// TIA Portal V19 export
FUNCTION_BLOCK "JB_FB"   // FB68, LAD
TITLE = JUNCTION BENCH WELDER
// stored: MemoryReserve 100, SetENOAutomatically false
   VAR_INPUT
      AreaInterface : "AreaInterface";
      ZSI : "udt_ZoneSafetyInterface";
      DSI : Struct
         Torch : "udt_DeviceSafetyInterface";
         ClampEntry : "udt_DeviceSafetyInterface";
         ClampExit : "udt_DeviceSafetyInterface";
         CutHead : "udt_DeviceSafetyInterface";
         PinchRoll_Feed : "udt_DeviceSafetyInterface";
         PinchRoll_Lift : "udt_DeviceSafetyInterface";
      END_STRUCT;
      Drive : Struct
         Torch : "TAx_DriveInterface";
         Picnhroll_Feed : "TAx_DriveInterface";
      END_STRUCT;
      HWID : Struct
         Torch_TEL1 : HW_SUBMODULE;
         TorchEnc_IO : HW_SUBMODULE;
         Pinchroll_Feed_TEL1 : HW_SUBMODULE;
      END_STRUCT;
      DataIn : Struct
         WeldingCycle_AI_Potentiometer : Int;
         WeldingCycle_Pb_Stop : Bool;
         WeldingCycle_Pb_Start : Bool;
         WeldingCycle_Pb_StartStop : Bool;
         Welder_Pb_Man : Bool;
         CutHead_PbCycle : Bool;
         SAFETY_DeadMan_PB : Bool;   // Pulsante presenza uomo SAFTEY
         Torch : "Positioning_DOL_Machine_DataIn";
         ClampEntry : "ValveMachine_DataIn";
         ClampExit : "ValveMachine_DataIn";
         CutHead : "ValveMachine_DataIn";
         PinchRoll_Feed : "SpeedMachine_DataIn";
         PinchRoll_Lift : "ValveMachine_DataIn";
      END_STRUCT;
      CIn : Struct
         Manager : "JB_Manager";
         PressureRunning : Bool;
      END_STRUCT;
      Config : Struct
         MeasurePasslineReference : Real;   // Distance of sheet passline from reference
         MaxMaterialWidth : Real;
         Torch : "Positioning_DOL_Machine_Config";
         ClampEntry : "ValveMachine_Config";
         ClampExit : "ValveMachine_Config";
         CutHead : "ValveMachine_Config";
         Pinchroll_Feed : "SpeedMachine_Config";
         Pinchroll_Lift : "ValveMachine_Config";
      END_STRUCT;
   END_VAR
   VAR_OUTPUT
      MachineInterface : "MachineInterface";
      DataOut : Struct
         LpWeldingCycle_1 : Bool;   // Lamp cmd of weldong cycle started inside the guards
         LpWeldingCycle_2 : Bool;   // Lamp cmd of weldong cycle started outside the guards
         WelderON : Bool;
         AspiratoreON : Bool;
         Torch : "Positioning_DOL_Machine_DataOut";
         ClampEntry : "ValveMachine_DataOut";
         ClampExit : "ValveMachine_DataOut";
         CutHead : "ValveMachine_DataOut";
         Pinchroll_Feed : "SpeedMachine_DataOut";
         Pinchroll_Lift : "ValveMachine_DataOut";
      END_STRUCT;
      COut : "JB_Status";
   END_VAR
   VAR_IN_OUT
      PersistentValues : Struct
         Data : Struct
            WeldingSetUp : "JB_WeldingSetUp";
            ClampEntryClosed : Bool;
            ClampExitClosed : Bool;
         END_STRUCT;
         Torch : Struct
            MeasureTorchHolder : LReal;   // Distance from sliding block & torch holder
            InhibitWeld_Pos : LReal;
            InhibitWeld_Window : LReal;   // if > 0 the ihhibit is enabled
            Parking_Pos : LReal;
            WeldingUseLocalData : Bool;   // TRUE = USE LOCAL DATA / FALSE = USE PROFILE DATA
            Cycle_HighSpeed : LReal;   // 0..100%
            Cycle_LowSpeed : LReal;   // 0..100%
         END_STRUCT;
         TorchAx : "Positioning_DOL_Machine_Par";
         TorchAx_Pers : "Positioning_DOL_Machine_Pers_Data";
         TorchEnc : "PosFbk_RTN";
         PinchRoll_Feed : "SpeedMachine_Par";
         Aspiratore_TimeOff : Time;
      END_STRUCT;
   END_VAR
   VAR
      Alarm : Struct
         TorchAx : "Positioning_DOL_Machine_Alr";
         TorchEnc : "PosFbk_Encoder_Alr";
         ClampEntry : "ValveAlr";
         ClampExit : "ValveAlr";
         CutHead : "ValveAlr";
         Pinchroll_Feed : "SpeedMachine_Alr";
         Pinchroll_Lift : "ValveAlr";
      END_STRUCT;
      Warning : Struct
         TorchAx : "Positioning_DOL_Machine_Wng";
         ClampEntry : "ValveMachine_Wng";
         ClampExit : "ValveMachine_Wng";
         CutHead : "ValveMachine_Wng";
         Pinchroll_Feed : "SpeedMachine_Wng";
         Pinchroll_Lift : "ValveMachine_Wng";
      END_STRUCT;
      HMI : Struct
         Torch_B_Preset : Bool;
         Torch_PresetValue : LReal;
         Torch_FdbkPreset : LReal;
      END_STRUCT;
      Sts : Struct
         Torch : Struct
            InParkPosition : Bool;
            InOutEdgeOfWeldStart : Bool;
            InWeldStart : Bool;
            inWeldStop : Bool;
            InPotentimeterON : Bool;
            InWeldON : Bool;
            InWeldInhibit : Bool;
         END_STRUCT;
         WeldCycle : Struct
            Phase : Int;
            Cnd : Bool;
            ON1 : Bool;   // 1 = Start form button inside guards
            ON2 : Bool;   // 2 = Start from button outside guards
            PercentagePotentiometer : Real;
            PosOutStripEdgeSideWeldStart : LReal;   // Position 5 mm out of the strip edge used as welding start
            PosOutStripEdgeSideWeldStop : LReal;
            PosStripEdgeSideWeldStart : LReal;
            PosStripEdgeSideWeldStop : LReal;
            PosWeldStart : LReal;   // Position of weld start (inside the entry strip edge)
            PosWeldStop : LReal;   // Position of weld stop (inside the exit strip edge)
            PosMinusInhibit : LReal;   // Limit minus where Inhibi the welding in order to skip the hole for referenced the junctio position
            PosPlusInhibit : LReal;   // Limit plus where Inhibi the welding in order to skip the hole for referenced the junctio position
            TON_Pause { S7_SetPoint := 'True'} : TON_TIME;
         END_STRUCT;
         CutCycle : Struct
            ON : Bool;
            OK_Rest : Bool;
            OK_Work : Bool;
         END_STRUCT;
      END_STRUCT;
      Ctrl : Struct
         WeldCycle : Struct
            Clamps_Close : Bool;
            Clamps_Open : Bool;
            Welder_ON : Bool;
            Torch_MoveToPos_Park : Bool;
            Torch_MoveToPos_Start : Bool;
            Torch_MoveToPos_StartBack : Bool;
            Torch_VelBwd_WeldON : Bool;
            Torch_VelFwd_WeldON : Bool;
         END_STRUCT;
         Welder : Struct
            Man_ON : Bool;
         END_STRUCT;
      END_STRUCT;
      Torch : "Positioning_DOL_Machine_FB";
      TorchEnc : "PosFbk_SickANM58";
      TorchEncITF : "PosFbk_ITF";
      ClampEntry : "ValveMachine_FB";
      ClampExit : "ValveMachine_FB";
      CutHead : "ValveMachine_FB";
      PinchRoll_Feed : "SpeedMachine_FB";
      PinchRoll_Lift : "ValveMachine_FB";
      TON_LiftPbUp : TON_TIME;
      TOF_Aspiratore { S7_SetPoint := 'True'} : TOF_TIME;
      AUX : Struct
         PbStartStop { ExternalAccessible := 'False'; ExternalVisible := 'False'; ExternalWritable := 'False'} : Bool;
         PbStart2 : Bool;
         Welder_Pb_Man : Bool;
         UseDataPPrf : Bool;
         Weld_PbCycle : Bool;
         Cut_PbCycle : Bool;
      END_STRUCT;
   END_VAR
   VAR_TEMP
      PE : Struct
         Weld_PbStartStop : Bool;
         Weld_PbStart1 : Bool;
         Weld_PStop1 : Bool;
         Weld_PbStart2 : Bool;
         Cut_PbCycle : Bool;
      END_STRUCT;
      CurrentWeldingSetUp : "JB_WeldingSetUp";
      PosOK : Bool;
      ParkPosPositiveSign : Bool;
      CndWelderON : Bool;
      retVal : Int;
      MaterialWidth : LReal;
      HalfMaterialWidth : LReal;
      MaterialOffset : LReal;
      HalfInhibitWindow : LReal;
      Stop : Bool;
      Pb_Rest : Bool;
      Pb_Work : Bool;
   END_VAR
   VAR CONSTANT
      PHASE_00_IDLE : Int := 0;
      PHASE_01_CLAMPS_CLOSE : Int := 1;
      PHASE_02_MOVE_TO_WELD_START : Int := 2;
      PHASE_03_WAIT_START_ACK : Int := 3;
      PHASE_04_MOVE_TORCH_OUT_STRIP : Int := 4;
      PHASE_05_MOVE_VELCITY_AND_WELDING : Int := 5;
      PHASE_06_WIAT_2SEC_AFTER_WELDING : Int := 6;
      PHASE_07_MOVE_TO_PARKING : Int := 7;
      PHASE_08_CLAMPS_OPEN : Int := 8;
   END_VAR
   VAR_TEMP   // added for the SCL form of the ladder/FBD networks
      _w1 : Bool;
      _w2 : Bool;
   END_VAR
BEGIN

REGION Network 1: <<< WELDING CYCLE >>>>
END_REGION

REGION Network 2: Welding velocity by scaling potentiometer
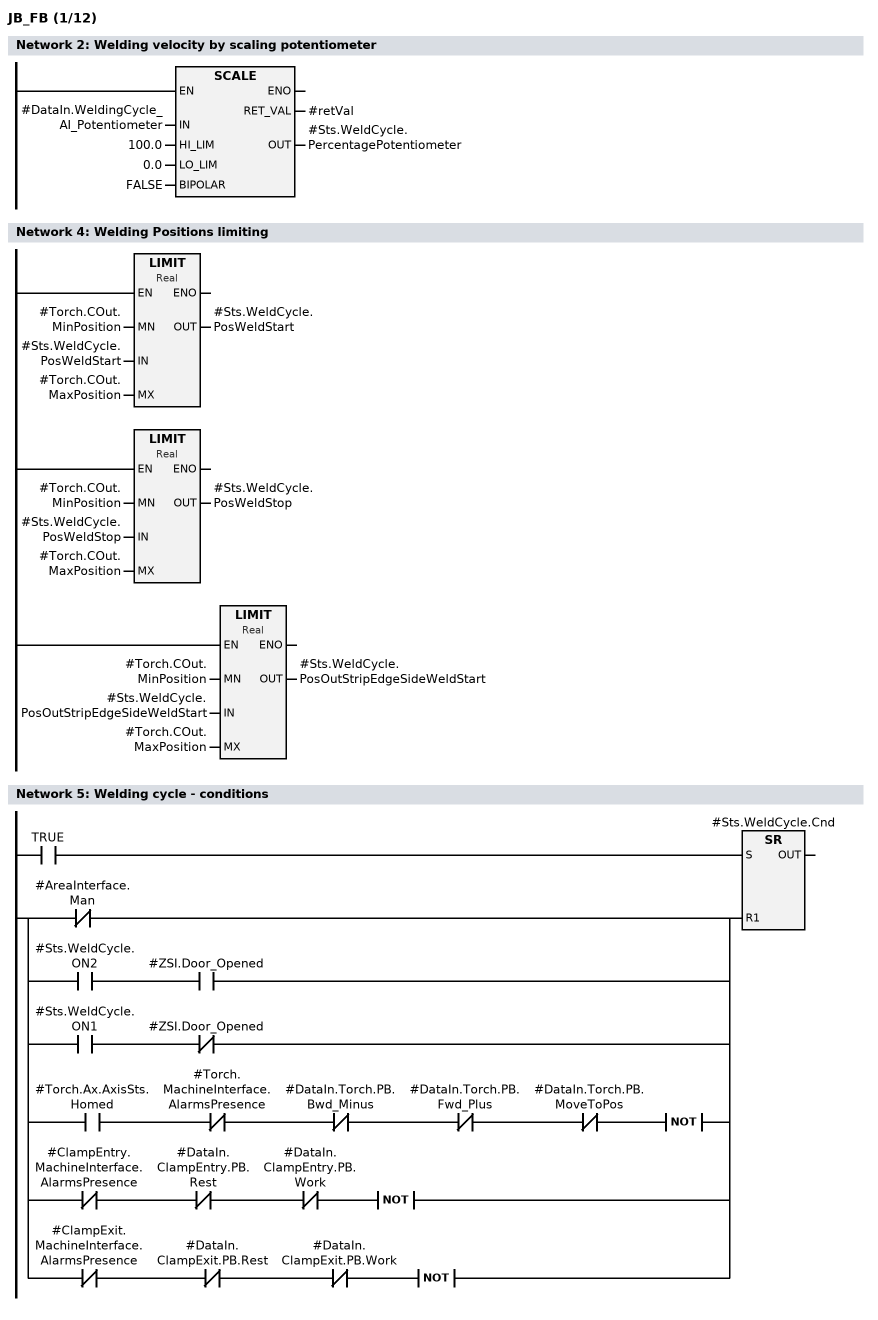
   #retVal := SCALE(IN := #DataIn.WeldingCycle_AI_Potentiometer,
                    HI_LIM := 100.0,
                    LO_LIM := 0.0,
                    BIPOLAR := FALSE,
                    OUT => #Sts.WeldCycle.PercentagePotentiometer);
END_REGION

REGION Network 3 (SCL): Welding Positions calculations
   // Switch between profile data & local data
   // 
   IF #PersistentValues.Torch.WeldingUseLocalData THEN

       IF  #AUX.UseDataPPrf THEN

           #PersistentValues.Data.WeldingSetUp := #CIn.Manager.WeldingSetUp;
       END_IF;

       #AUX.UseDataPPrf := FALSE;

       #CurrentWeldingSetUp := #PersistentValues.Data.WeldingSetUp ;


   ELSE
       #AUX.UseDataPPrf := TRUE;
       #CurrentWeldingSetUp := #CIn.Manager.WeldingSetUp;

   END_IF;



   // Material width
   // 
   #MaterialWidth := #Config.MaxMaterialWidth;

   IF #CurrentWeldingSetUp.MaterialWidth > 0.0
   THEN
       #MaterialWidth := #CurrentWeldingSetUp.MaterialWidth;
   END_IF;

   #MaterialWidth := MIN(IN1 := #Config.MaxMaterialWidth, IN2 := #MaterialWidth);

   #HalfMaterialWidth := #MaterialWidth / 2;


   // Material offset
   // 
   IF #CurrentWeldingSetUp.MeasureSheetEdgeReference <= 0.0
   THEN
       #MaterialOffset := 0.0;
   ELSE
       #MaterialOffset := - (#Config.MeasurePasslineReference - ABS(#CurrentWeldingSetUp.MeasureSheetEdgeReference) - #HalfMaterialWidth);
   END_IF;


   // Park position is positive = The parking position is away from operator = in the motor side
   // if is negative the parking is near the operator side
   //
   #ParkPosPositiveSign := #PersistentValues.Torch.Parking_Pos > 0.0;



   // Welding cam track case Direction is from BKW=Minus (op.side) to FWD=Plus (motor side) 
   // 


   IF #CurrentWeldingSetUp.WeldingDirection THEN


       #Sts.WeldCycle.PosStripEdgeSideWeldStart := - #HalfMaterialWidth + #MaterialOffset;
       #Sts.WeldCycle.PosStripEdgeSideWeldStop := #HalfMaterialWidth + #MaterialOffset;

       #Sts.WeldCycle.PosWeldStart := #Sts.WeldCycle.PosStripEdgeSideWeldStart +  #CurrentWeldingSetUp.CorrStartWelding;
       #Sts.WeldCycle.PosWeldStop := #Sts.WeldCycle.PosStripEdgeSideWeldStop - #CurrentWeldingSetUp.CorrStopWelding;

       #Sts.WeldCycle.PosOutStripEdgeSideWeldStart := #Sts.WeldCycle.PosStripEdgeSideWeldStart - 5.0;
       #Sts.WeldCycle.PosOutStripEdgeSideWeldStop := #Sts.WeldCycle.PosStripEdgeSideWeldStart + 5.0;


   END_IF;


   // Welding cam track case Direction is from FWD (motor side) to BKD (op.side)
   // 
   IF NOT #CurrentWeldingSetUp.WeldingDirection THEN


       #Sts.WeldCycle.PosStripEdgeSideWeldStart := #HalfMaterialWidth + #MaterialOffset;
       #Sts.WeldCycle.PosStripEdgeSideWeldStop := - #HalfMaterialWidth + #MaterialOffset;

       #Sts.WeldCycle.PosWeldStart := #Sts.WeldCycle.PosStripEdgeSideWeldStart - #CurrentWeldingSetUp.CorrStartWelding;
       #Sts.WeldCycle.PosWeldStop := #Sts.WeldCycle.PosStripEdgeSideWeldStop + #CurrentWeldingSetUp.CorrStopWelding;

       #Sts.WeldCycle.PosOutStripEdgeSideWeldStart := #Sts.WeldCycle.PosStripEdgeSideWeldStart + 5.0;
       #Sts.WeldCycle.PosOutStripEdgeSideWeldStop := #Sts.WeldCycle.PosStripEdgeSideWeldStart - 5.0;

   END_IF;


   // // Welding Inhibit zone
   // 
   #HalfInhibitWindow := #PersistentValues.Torch.InhibitWeld_Window / 2.0;
   #Sts.WeldCycle.PosMinusInhibit := #PersistentValues.Torch.InhibitWeld_Pos - #HalfInhibitWindow + #MaterialOffset;
   #Sts.WeldCycle.PosPlusInhibit := #PersistentValues.Torch.InhibitWeld_Pos + #HalfInhibitWindow + #MaterialOffset;
END_REGION

REGION Network 4: Welding Positions limiting
   RUNG wire#powerrail
      { S7_Templates := "value_type := Real" } Limit(mn := #Torch.COut.MinPosition, in := #Sts.WeldCycle.PosWeldStart, mx := #Torch.COut.MaxPosition, out => #Sts.WeldCycle.PosWeldStart)
   END_RUNG
   RUNG wire#powerrail
      { S7_Templates := "value_type := Real" } Limit(mn := #Torch.COut.MinPosition, in := #Sts.WeldCycle.PosWeldStop, mx := #Torch.COut.MaxPosition, out => #Sts.WeldCycle.PosWeldStop)
   END_RUNG
   RUNG wire#powerrail
      { S7_Templates := "value_type := Real" } Limit(mn := #Torch.COut.MinPosition, in := #Sts.WeldCycle.PosOutStripEdgeSideWeldStart, mx := #Torch.COut.MaxPosition, out => #Sts.WeldCycle.PosOutStripEdgeSideWeldStart)
   END_RUNG
   // the same network as SCL:
   #Sts.WeldCycle.PosWeldStart := LIMIT(MN := #Torch.COut.MinPosition, IN := #Sts.WeldCycle.PosWeldStart, MX := #Torch.COut.MaxPosition);
   #Sts.WeldCycle.PosWeldStop := LIMIT(MN := #Torch.COut.MinPosition, IN := #Sts.WeldCycle.PosWeldStop, MX := #Torch.COut.MaxPosition);
   #Sts.WeldCycle.PosOutStripEdgeSideWeldStart := LIMIT(MN := #Torch.COut.MinPosition, IN := #Sts.WeldCycle.PosOutStripEdgeSideWeldStart, MX := #Torch.COut.MaxPosition);
END_REGION

REGION Network 5: Welding cycle - conditions
   RUNG wire#powerrail
      Contact( TRUE )
      S_SR(operand := #Sts.WeldCycle.Cnd, r1 := wire#w1)
   END_RUNG
   RUNG wire#powerrail
      I_Contact( #AreaInterface.Man )
   END_RUNG wire#w1
   RUNG wire#powerrail
      Contact( #Sts.WeldCycle.ON2 )
      Contact( #ZSI.Door_Opened )
   END_RUNG wire#w1
   RUNG wire#powerrail
      Contact( #Sts.WeldCycle.ON1 )
      I_Contact( #ZSI.Door_Opened )
   END_RUNG wire#w1
   RUNG wire#powerrail
      Contact( #Torch.Ax.AxisSts.Homed )
      I_Contact( #Torch.MachineInterface.AlarmsPresence )
      I_Contact( #DataIn.Torch.PB.Bwd_Minus )
      I_Contact( #DataIn.Torch.PB.Fwd_Plus )
      I_Contact( #DataIn.Torch.PB.MoveToPos )
      Not()
   END_RUNG wire#w1
   RUNG wire#powerrail
      I_Contact( #ClampEntry.MachineInterface.AlarmsPresence )
      I_Contact( #DataIn.ClampEntry.PB.Rest )
      I_Contact( #DataIn.ClampEntry.PB.Work )
      Not()
   END_RUNG wire#w1
   RUNG wire#powerrail
      I_Contact( #ClampExit.MachineInterface.AlarmsPresence )
      I_Contact( #DataIn.ClampExit.PB.Rest )
      I_Contact( #DataIn.ClampExit.PB.Work )
      Not()
   END_RUNG wire#w1
   // the same network as SCL:
   IF TRUE THEN
       #Sts.WeldCycle.Cnd := TRUE;   // SR flip-flop
   END_IF;
   IF NOT #AreaInterface.Man OR (#Sts.WeldCycle.ON2 AND #ZSI.Door_Opened) OR (#Sts.WeldCycle.ON1 AND NOT #ZSI.Door_Opened) OR NOT (#Torch.Ax.AxisSts.Homed AND NOT #Torch.MachineInterface.AlarmsPresence AND NOT #DataIn.Torch.PB.Bwd_Minus AND NOT #DataIn.Torch.PB.Fwd_Plus AND NOT #DataIn.Torch.PB.MoveToPos) OR NOT (NOT #ClampEntry.MachineInterface.AlarmsPresence AND NOT #DataIn.ClampEntry.PB.Rest AND NOT #DataIn.ClampEntry.PB.Work) OR NOT (NOT #ClampExit.MachineInterface.AlarmsPresence AND NOT #DataIn.ClampExit.PB.Rest AND NOT #DataIn.ClampExit.PB.Work) THEN
       #Sts.WeldCycle.Cnd := FALSE;
   END_IF;
END_REGION

REGION Network 6: Welding cycle - Start / Stop
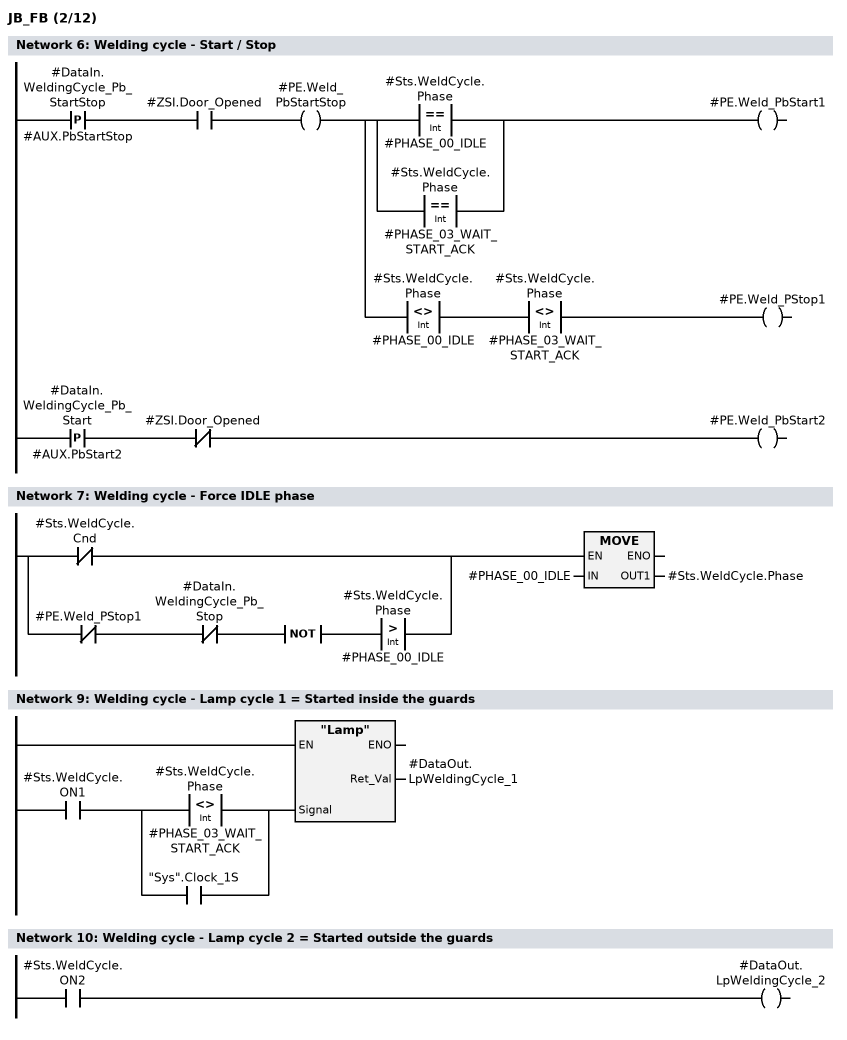
   RUNG wire#powerrail
      P_Contact(operand := #DataIn.WeldingCycle_Pb_StartStop, bit := #AUX.PbStartStop)
      Contact( #ZSI.Door_Opened )
      Coil( #PE.Weld_PbStartStop )
      wire#w1
      { S7_Templates := "SrcType := Int" } EQ_Contact(in1 := #Sts.WeldCycle.Phase, in2 := #PHASE_00_IDLE)
      wire#w2
      Coil( #PE.Weld_PbStart1 )
   END_RUNG
   RUNG wire#w1
      { S7_Templates := "SrcType := Int" } EQ_Contact(in1 := #Sts.WeldCycle.Phase, in2 := #PHASE_03_WAIT_START_ACK)
   END_RUNG wire#w2
   RUNG wire#w1
      { S7_Templates := "SrcType := Int" } NE_Contact(in1 := #Sts.WeldCycle.Phase, in2 := #PHASE_00_IDLE)
      { S7_Templates := "SrcType := Int" } NE_Contact(in1 := #Sts.WeldCycle.Phase, in2 := #PHASE_03_WAIT_START_ACK)
      Coil( #PE.Weld_PStop1 )
   END_RUNG
   RUNG wire#powerrail
      P_Contact(operand := #DataIn.WeldingCycle_Pb_Start, bit := #AUX.PbStart2)
      I_Contact( #ZSI.Door_Opened )
      Coil( #PE.Weld_PbStart2 )
   END_RUNG
   // the same network as SCL:
   #_w1 := #DataIn.WeldingCycle_Pb_StartStop AND NOT #AUX.PbStartStop;   // rising edge of #DataIn.WeldingCycle_Pb_StartStop
   #AUX.PbStartStop := #DataIn.WeldingCycle_Pb_StartStop;
   #PE.Weld_PbStartStop := #_w1 AND #ZSI.Door_Opened;
   #PE.Weld_PbStart1 := #PE.Weld_PbStartStop AND ((#Sts.WeldCycle.Phase = #PHASE_00_IDLE) OR (#Sts.WeldCycle.Phase = #PHASE_03_WAIT_START_ACK));
   #PE.Weld_PStop1 := #PE.Weld_PbStartStop AND (#Sts.WeldCycle.Phase <> #PHASE_00_IDLE) AND (#Sts.WeldCycle.Phase <> #PHASE_03_WAIT_START_ACK);
   #_w2 := #DataIn.WeldingCycle_Pb_Start AND NOT #AUX.PbStart2;   // rising edge of #DataIn.WeldingCycle_Pb_Start
   #AUX.PbStart2 := #DataIn.WeldingCycle_Pb_Start;
   #PE.Weld_PbStart2 := #_w2 AND NOT #ZSI.Door_Opened;
END_REGION

REGION Network 7: Welding cycle - Force IDLE phase
   RUNG wire#powerrail
      I_Contact( #Sts.WeldCycle.Cnd )
      wire#w1
      { S7_GenerateENO := "TRUE" } Move(in := #PHASE_00_IDLE, out1 => #Sts.WeldCycle.Phase)
   END_RUNG
   RUNG wire#powerrail
      I_Contact( #PE.Weld_PStop1 )
      I_Contact( #DataIn.WeldingCycle_Pb_Stop )
      Not()
      { S7_Templates := "SrcType := Int" } GT_Contact(in1 := #Sts.WeldCycle.Phase, in2 := #PHASE_00_IDLE)
   END_RUNG wire#w1
   // the same network as SCL:
   IF NOT #Sts.WeldCycle.Cnd OR (NOT (NOT #PE.Weld_PStop1 AND NOT #DataIn.WeldingCycle_Pb_Stop) AND (#Sts.WeldCycle.Phase > #PHASE_00_IDLE)) THEN
       #Sts.WeldCycle.Phase := #PHASE_00_IDLE;
   END_IF;
END_REGION

REGION Network 8 (SCL): Welding cycle - Sequence
   CASE #Sts.WeldCycle.Phase OF




       //############################################################################################
       // PHASE 00 - IDLE
       //############################################################################################
       //    
       #PHASE_00_IDLE:

           #Sts.WeldCycle.ON1 := FALSE;
           #Sts.WeldCycle.ON2 := FALSE;


           #Sts.WeldCycle.TON_Pause(IN:=FALSE,PT:=T#2s);

           #Ctrl.WeldCycle.Clamps_Close := FALSE;
           #Ctrl.WeldCycle.Clamps_Open := FALSE;
           #Ctrl.WeldCycle.Welder_ON := FALSE;
           #Ctrl.WeldCycle.Torch_MoveToPos_Park := FALSE;
           #Ctrl.WeldCycle.Torch_MoveToPos_Start := FALSE;
           #Ctrl.WeldCycle.Torch_MoveToPos_StartBack := FALSE;
           #Ctrl.WeldCycle.Torch_VelBwd_WeldON := FALSE;
           #Ctrl.WeldCycle.Torch_VelFwd_WeldON := FALSE;


           IF #PE.Weld_PbStart1 THEN

               #Sts.WeldCycle.ON1 := TRUE;

               #Sts.WeldCycle.Phase +=1;
           END_IF;


           IF #PE.Weld_PbStart2 THEN

               #Sts.WeldCycle.ON2 := TRUE;

               #Sts.WeldCycle.Phase +=1;
           END_IF;





       //############################################################################################
       // PHASE 01 - CLOSE CLAMPS
       //############################################################################################
       //
       #PHASE_01_CLAMPS_CLOSE:


           #Ctrl.WeldCycle.Clamps_Close := NOT #ClampEntry.V.ValveSts.IsAtWork OR NOT #ClampExit.V.ValveSts.IsAtWork;

           IF NOT #Ctrl.WeldCycle.Clamps_Close THEN

               // New start or restart?
               // 
               // Se il ciclo è avviato con la torcia già nel range di saldatura non si passa per la fase di la conferma della regolazione (Verticale / Longitudinale) della torcia.
               // 
               // Questa condizione si verifica se durante la saldtaura si è interrotto il ciclo (rilascio pulsante di abilitazione + comando avanti o indietro torcia)
               // e successiva ripartenza del ciclo di saldatura..
               // 
               IF NOT #Sts.Torch.InWeldON THEN
                   #Sts.WeldCycle.Phase +=1;
               ELSE
                   #Sts.WeldCycle.Phase := #PHASE_05_MOVE_VELCITY_AND_WELDING;
               END_IF;
           END_IF;


       //############################################################################################
       // PHASE 02 - MOVE TORCH TO WELD START
       //############################################################################################ 
       //
       #PHASE_02_MOVE_TO_WELD_START :

           #Ctrl.WeldCycle.Torch_MoveToPos_Start := NOT #Sts.Torch.InWeldStart;

           IF NOT #Ctrl.WeldCycle.Torch_MoveToPos_Start THEN
               #Sts.WeldCycle.Phase +=1;
           END_IF;



       //############################################################################################
       // PHASE 03 - WAIT ACK TO START THE WELDNG
       //############################################################################################   
       //
       #PHASE_03_WAIT_START_ACK :

           // Attesa della nuova pressione del pulsante di start per confermare che la regolazione verticale e longitudinale della torcia sono state
           // eseguite e quindi la sa

           IF #PE.Weld_PbStart1 OR #Sts.WeldCycle.ON2  THEN
               #Sts.WeldCycle.Phase +=1;
           END_IF;



       //############################################################################################
       // PHASE 04 - MOVE TORCH OUT OF THE STRIP EDGE USED AS WELDING START
       //############################################################################################
       //
       #PHASE_04_MOVE_TORCH_OUT_STRIP :

           #Ctrl.WeldCycle.Torch_MoveToPos_StartBack := NOT #Sts.Torch.InOutEdgeOfWeldStart;

           IF NOT #Ctrl.WeldCycle.Torch_MoveToPos_StartBack THEN
               #Sts.WeldCycle.Phase +=1;
           END_IF;



       //############################################################################################
       // PHASE 05 - MOVE TORCH VELOCITY AND START WELDING 
       //############################################################################################
       //
       #PHASE_05_MOVE_VELCITY_AND_WELDING :

           #Ctrl.WeldCycle.Torch_VelBwd_WeldON := NOT #Sts.Torch.inWeldStop AND NOT #CurrentWeldingSetUp.WeldingDirection;
           #Ctrl.WeldCycle.Torch_VelFwd_WeldON := NOT #Sts.Torch.inWeldStop AND #CurrentWeldingSetUp.WeldingDirection;

           #Ctrl.WeldCycle.Welder_ON := NOT #Sts.Torch.inWeldStop AND NOT #Sts.Torch.InWeldInhibit;

           IF NOT #Ctrl.WeldCycle.Torch_VelBwd_WeldON AND NOT #Ctrl.WeldCycle.Torch_VelFwd_WeldON AND NOT #Ctrl.WeldCycle.Welder_ON  THEN

               #Sts.WeldCycle.TON_Pause(IN:=FALSE,PT:=T#2s);
               #Sts.WeldCycle.Phase +=1;
           END_IF;


       //############################################################################################
       // PHASE 06 - WAIT 2 SECONDS
       //############################################################################################   
       //

       #PHASE_06_WIAT_2SEC_AFTER_WELDING :

           #Sts.WeldCycle.TON_Pause(IN:=TRUE,PT:=T#2s);

           IF #Sts.WeldCycle.TON_Pause.Q THEN
               #Sts.WeldCycle.Phase +=1;
           END_IF;


       //############################################################################################
       // PHASE 07 - MOVE TORCH TO PARKING POSITION
       //############################################################################################
       //
       #PHASE_07_MOVE_TO_PARKING:

           #Ctrl.WeldCycle.Torch_MoveToPos_Park := NOT #Sts.Torch.InParkPosition;

           IF NOT #Ctrl.WeldCycle.Torch_MoveToPos_Park THEN
               #Sts.WeldCycle.Phase +=1;
           END_IF;



       //############################################################################################
       // PHASE 08 - CLAMPS OPEN
       //############################################################################################
       //
       #PHASE_08_CLAMPS_OPEN :

           #Ctrl.WeldCycle.Clamps_Open := NOT #ClampEntry.V.ValveSts.IsAtRest OR NOT #ClampExit.V.ValveSts.IsAtRest;

           IF NOT  #Ctrl.WeldCycle.Clamps_Open THEN

               #Sts.WeldCycle.Phase := 0;

           END_IF;




       ELSE
           #Sts.WeldCycle.Phase := 0;



       END_CASE;
END_REGION

REGION Network 9: Welding cycle - Lamp cycle 1 = Started inside the guards
   RUNG wire#powerrail
      "Lamp"(Signal := wire#w2, Ret_Val => #DataOut.LpWeldingCycle_1)
   END_RUNG
   RUNG wire#powerrail
      Contact( #Sts.WeldCycle.ON1 )
      wire#w1
      { S7_Templates := "SrcType := Int" } NE_Contact(in1 := #Sts.WeldCycle.Phase, in2 := #PHASE_03_WAIT_START_ACK)
   END_RUNG wire#w2
   RUNG wire#w1
      Contact( "Sys".Clock_1S )
   END_RUNG wire#w2
   // the same network as SCL:
   #DataOut.LpWeldingCycle_1 := "Lamp"(Signal := #Sts.WeldCycle.ON1 AND ((#Sts.WeldCycle.Phase <> #PHASE_03_WAIT_START_ACK) OR "Sys".Clock_1S));
END_REGION

REGION Network 10: Welding cycle - Lamp cycle 2 = Started outside the guards
   RUNG wire#powerrail
      Contact( #Sts.WeldCycle.ON2 )
      Coil( #DataOut.LpWeldingCycle_2 )
   END_RUNG
   // the same network as SCL:
   #DataOut.LpWeldingCycle_2 := #Sts.WeldCycle.ON2;
END_REGION

REGION Network 11: >
END_REGION

REGION Network 12: >
END_REGION

REGION Network 13: >
END_REGION

REGION Network 14: <<< WELDER TORCH >>>
END_REGION

REGION Network 15: CIn (Manager = Welding cycle)
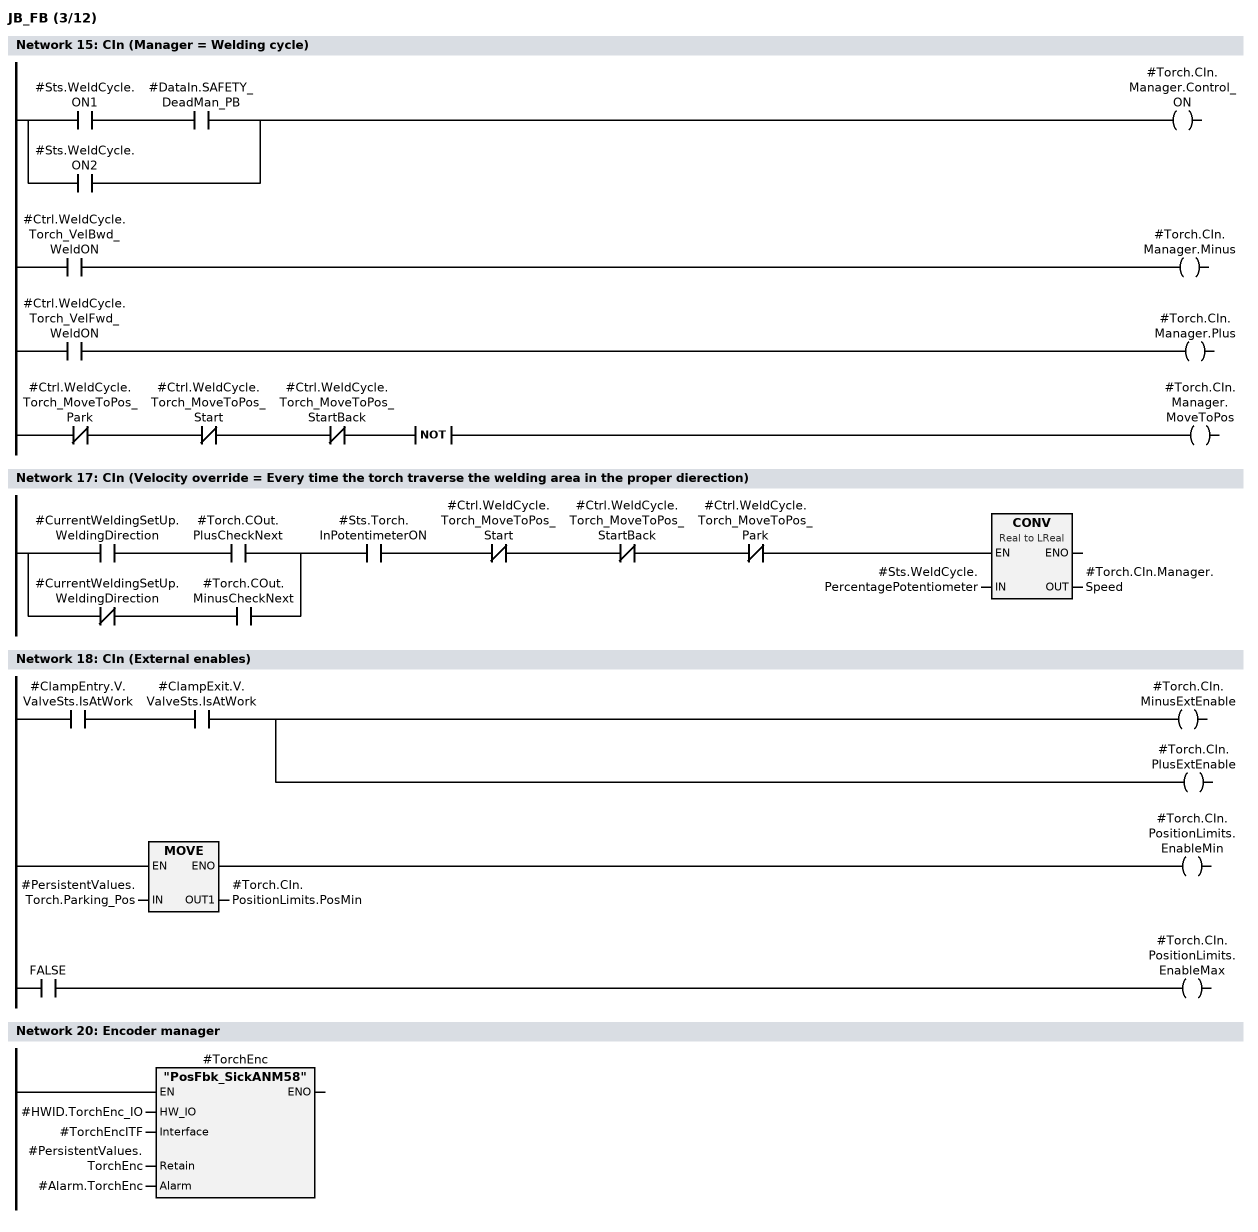
   RUNG wire#powerrail
      Contact( #Sts.WeldCycle.ON1 )
      Contact( #DataIn.SAFETY_DeadMan_PB )
      wire#w1
      Coil( #Torch.CIn.Manager.Control_ON )
   END_RUNG
   RUNG wire#powerrail
      Contact( #Sts.WeldCycle.ON2 )
   END_RUNG wire#w1
   RUNG wire#powerrail
      Contact( #Ctrl.WeldCycle.Torch_VelBwd_WeldON )
      Coil( #Torch.CIn.Manager.Minus )
   END_RUNG
   RUNG wire#powerrail
      Contact( #Ctrl.WeldCycle.Torch_VelFwd_WeldON )
      Coil( #Torch.CIn.Manager.Plus )
   END_RUNG
   RUNG wire#powerrail
      I_Contact( #Ctrl.WeldCycle.Torch_MoveToPos_Park )
      I_Contact( #Ctrl.WeldCycle.Torch_MoveToPos_Start )
      I_Contact( #Ctrl.WeldCycle.Torch_MoveToPos_StartBack )
      Not()
      Coil( #Torch.CIn.Manager.MoveToPos )
   END_RUNG
   // the same network as SCL:
   #Torch.CIn.Manager.Control_ON := (#Sts.WeldCycle.ON1 AND #DataIn.SAFETY_DeadMan_PB) OR #Sts.WeldCycle.ON2;
   #Torch.CIn.Manager.Minus := #Ctrl.WeldCycle.Torch_VelBwd_WeldON;
   #Torch.CIn.Manager.Plus := #Ctrl.WeldCycle.Torch_VelFwd_WeldON;
   #Torch.CIn.Manager.MoveToPos := NOT (NOT #Ctrl.WeldCycle.Torch_MoveToPos_Park AND NOT #Ctrl.WeldCycle.Torch_MoveToPos_Start AND NOT #Ctrl.WeldCycle.Torch_MoveToPos_StartBack);
END_REGION

REGION Network 16 (SCL): CIn (manager Pos,Vel,Acc,Dec,Jerk)
   #Torch.CIn.Manager.Speed := 0.0;

   IF #Ctrl.WeldCycle.Torch_MoveToPos_Park THEN
       #Torch.CIn.Manager.Pos := #PersistentValues.Torch.Parking_Pos;
       #Torch.CIn.Manager.Speed := #PersistentValues.Torch.Cycle_HighSpeed;

   ELSIF #Ctrl.WeldCycle.Torch_MoveToPos_Start THEN
       #Torch.CIn.Manager.Pos := #Sts.WeldCycle.PosWeldStart;
       #Torch.CIn.Manager.Speed := #PersistentValues.Torch.Cycle_HighSpeed;


   ELSIF #Ctrl.WeldCycle.Torch_MoveToPos_StartBack THEN
       #Torch.CIn.Manager.Pos := #Sts.WeldCycle.PosOutStripEdgeSideWeldStart;
       #Torch.CIn.Manager.Speed := #PersistentValues.Torch.Cycle_LowSpeed;


   ELSIF #Ctrl.WeldCycle.Torch_VelBwd_WeldON OR #Ctrl.WeldCycle.Torch_VelFwd_WeldON THEN
       #Torch.CIn.Manager.Speed := 95.0;

   END_IF;
END_REGION

REGION Network 17: CIn (Velocity override = Every time the torch traverse the welding area in the proper dierection)
   RUNG wire#powerrail
      Contact( #CurrentWeldingSetUp.WeldingDirection )
      Contact( #Torch.COut.PlusCheckNext )
      wire#w1
      Contact( #Sts.Torch.InPotentimeterON )
      I_Contact( #Ctrl.WeldCycle.Torch_MoveToPos_Start )
      I_Contact( #Ctrl.WeldCycle.Torch_MoveToPos_StartBack )
      I_Contact( #Ctrl.WeldCycle.Torch_MoveToPos_Park )
      { S7_Templates := "[SrcType := Real, DestType := LReal]" } Convert(in := #Sts.WeldCycle.PercentagePotentiometer, out => #Torch.CIn.Manager.Speed)
   END_RUNG
   RUNG wire#powerrail
      I_Contact( #CurrentWeldingSetUp.WeldingDirection )
      Contact( #Torch.COut.MinusCheckNext )
   END_RUNG wire#w1
   // the same network as SCL:
   IF ((#CurrentWeldingSetUp.WeldingDirection AND #Torch.COut.PlusCheckNext) OR (NOT #CurrentWeldingSetUp.WeldingDirection AND #Torch.COut.MinusCheckNext)) AND #Sts.Torch.InPotentimeterON AND NOT #Ctrl.WeldCycle.Torch_MoveToPos_Start AND NOT #Ctrl.WeldCycle.Torch_MoveToPos_StartBack AND NOT #Ctrl.WeldCycle.Torch_MoveToPos_Park THEN
       #Torch.CIn.Manager.Speed := REAL_TO_LREAL(#Sts.WeldCycle.PercentagePotentiometer);
   END_IF;
END_REGION

REGION Network 18: CIn (External enables)
   RUNG wire#powerrail
      Contact( #ClampEntry.V.ValveSts.IsAtWork )
      Contact( #ClampExit.V.ValveSts.IsAtWork )
      wire#w1
      Coil( #Torch.CIn.MinusExtEnable )
   END_RUNG
   RUNG wire#w1
      Coil( #Torch.CIn.PlusExtEnable )
   END_RUNG
   RUNG wire#powerrail
      { S7_GenerateENO := "TRUE" } Move(in := #PersistentValues.Torch.Parking_Pos, out1 => #Torch.CIn.PositionLimits.PosMin)
      Coil( #Torch.CIn.PositionLimits.EnableMin )
   END_RUNG
   RUNG wire#powerrail
      Contact( FALSE )
      Coil( #Torch.CIn.PositionLimits.EnableMax )
   END_RUNG
   // the same network as SCL:
   // ENO of a box is taken as its EN; it also drops when the box reports an error
   #Torch.CIn.MinusExtEnable := #ClampEntry.V.ValveSts.IsAtWork AND #ClampExit.V.ValveSts.IsAtWork;
   #Torch.CIn.PlusExtEnable := #Torch.CIn.MinusExtEnable;
   #Torch.CIn.PositionLimits.PosMin := #PersistentValues.Torch.Parking_Pos;
   #Torch.CIn.PositionLimits.EnableMin := TRUE;
   #Torch.CIn.PositionLimits.EnableMax := FALSE;
END_REGION

REGION Network 19 (SCL): HMI preset position
   #Torch.HMI.B_Preset := #HMI.Torch_B_Preset;

   #Torch.HMI.PresetPosition := ABS(#HMI.Torch_PresetValue) + #PersistentValues.Torch.MeasureTorchHolder - #Config.MeasurePasslineReference;

   #HMI.Torch_FdbkPreset := #Torch.COut.ActualPosition - #PersistentValues.Torch.MeasureTorchHolder + #Config.MeasurePasslineReference;
END_REGION

REGION Network 20: Encoder manager
   RUNG wire#powerrail
      #TorchEnc(HW_IO := #HWID.TorchEnc_IO, Interface := #TorchEncITF, Retain := #PersistentValues.TorchEnc, Alarm := #Alarm.TorchEnc)
   END_RUNG
   // the same network as SCL:
   #TorchEnc(HW_IO := #HWID.TorchEnc_IO,   // "PosFbk_SickANM58"
             Interface := #TorchEncITF,
             Retain := #PersistentValues.TorchEnc,
             Alarm := #Alarm.TorchEnc);
END_REGION

REGION Network 21: Axis Machine Manager
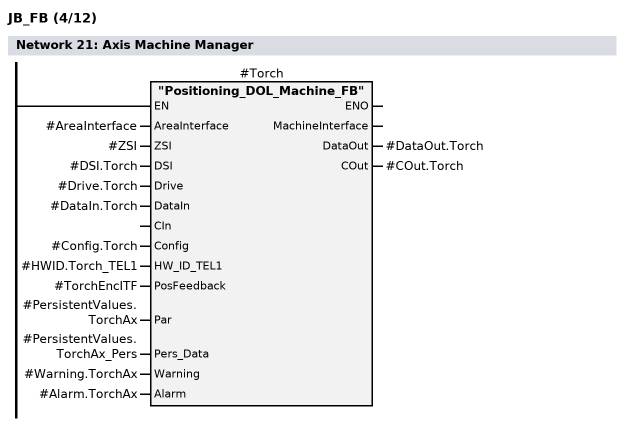
   RUNG wire#powerrail
      #Torch(AreaInterface := #AreaInterface, ZSI := #ZSI, DSI := #DSI.Torch, Drive := #Drive.Torch, DataIn := #DataIn.Torch, CIn :=, Config := #Config.Torch, HW_ID_TEL1 := #HWID.Torch_TEL1, PosFeedback := #TorchEncITF, Par := #PersistentValues.TorchAx, Pers_Data := #PersistentValues.TorchAx_Pers, Warning := #Warning.TorchAx, Alarm := #Alarm.TorchAx, MachineInterface =>, DataOut => #DataOut.Torch, COut => #COut.Torch)
   END_RUNG
   // the same network as SCL:
   #Torch(AreaInterface := #AreaInterface,   // "Positioning_DOL_Machine_FB"
          ZSI := #ZSI,
          DSI := #DSI.Torch,
          Drive := #Drive.Torch,
          DataIn := #DataIn.Torch,
          Config := #Config.Torch,
          HW_ID_TEL1 := #HWID.Torch_TEL1,
          PosFeedback := #TorchEncITF,
          Par := #PersistentValues.TorchAx,
          Pers_Data := #PersistentValues.TorchAx_Pers,
          Warning := #Warning.TorchAx,
          Alarm := #Alarm.TorchAx,
          DataOut => #DataOut.Torch,
          COut => #COut.Torch);
END_REGION

REGION Network 22: Torch positions status
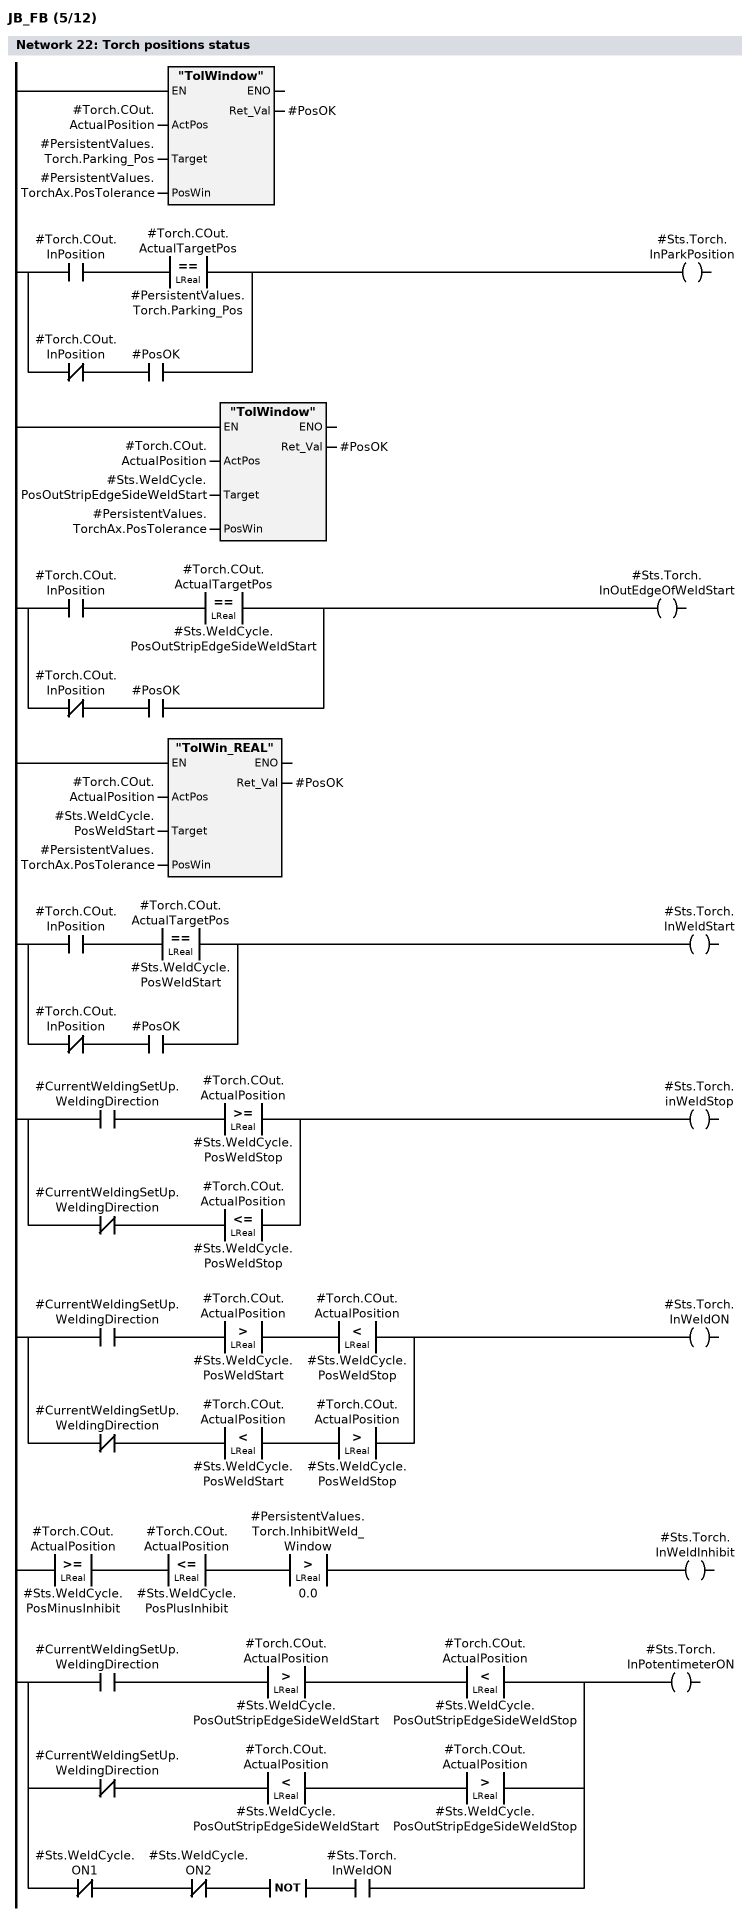
   RUNG wire#powerrail
      "TolWindow"(ActPos := #Torch.COut.ActualPosition, Target := #PersistentValues.Torch.Parking_Pos, PosWin := #PersistentValues.TorchAx.PosTolerance, Ret_Val => #PosOK)
   END_RUNG
   RUNG wire#powerrail
      Contact( #Torch.COut.InPosition )
      { S7_Templates := "SrcType := LReal" } EQ_Contact(in1 := #Torch.COut.ActualTargetPos, in2 := #PersistentValues.Torch.Parking_Pos)
      wire#w1
      Coil( #Sts.Torch.InParkPosition )
   END_RUNG
   RUNG wire#powerrail
      I_Contact( #Torch.COut.InPosition )
      Contact( #PosOK )
   END_RUNG wire#w1
   RUNG wire#powerrail
      "TolWindow"(ActPos := #Torch.COut.ActualPosition, Target := #Sts.WeldCycle.PosOutStripEdgeSideWeldStart, PosWin := #PersistentValues.TorchAx.PosTolerance, Ret_Val => #PosOK)
   END_RUNG
   RUNG wire#powerrail
      Contact( #Torch.COut.InPosition )
      { S7_Templates := "SrcType := LReal" } EQ_Contact(in1 := #Torch.COut.ActualTargetPos, in2 := #Sts.WeldCycle.PosOutStripEdgeSideWeldStart)
      wire#w2
      Coil( #Sts.Torch.InOutEdgeOfWeldStart )
   END_RUNG
   RUNG wire#powerrail
      I_Contact( #Torch.COut.InPosition )
      Contact( #PosOK )
   END_RUNG wire#w2
   RUNG wire#powerrail
      "TolWin_REAL"(ActPos := #Torch.COut.ActualPosition, Target := #Sts.WeldCycle.PosWeldStart, PosWin := #PersistentValues.TorchAx.PosTolerance, Ret_Val => #PosOK)
   END_RUNG
   RUNG wire#powerrail
      Contact( #Torch.COut.InPosition )
      { S7_Templates := "SrcType := LReal" } EQ_Contact(in1 := #Torch.COut.ActualTargetPos, in2 := #Sts.WeldCycle.PosWeldStart)
      wire#w3
      Coil( #Sts.Torch.InWeldStart )
   END_RUNG
   RUNG wire#powerrail
      I_Contact( #Torch.COut.InPosition )
      Contact( #PosOK )
   END_RUNG wire#w3
   RUNG wire#powerrail
      Contact( #CurrentWeldingSetUp.WeldingDirection )
      { S7_Templates := "SrcType := LReal" } GE_Contact(in1 := #Torch.COut.ActualPosition, in2 := #Sts.WeldCycle.PosWeldStop)
      wire#w4
      Coil( #Sts.Torch.inWeldStop )
   END_RUNG
   RUNG wire#powerrail
      I_Contact( #CurrentWeldingSetUp.WeldingDirection )
      { S7_Templates := "SrcType := LReal" } LE_Contact(in1 := #Torch.COut.ActualPosition, in2 := #Sts.WeldCycle.PosWeldStop)
   END_RUNG wire#w4
   RUNG wire#powerrail
      Contact( #CurrentWeldingSetUp.WeldingDirection )
      { S7_Templates := "SrcType := LReal" } GT_Contact(in1 := #Torch.COut.ActualPosition, in2 := #Sts.WeldCycle.PosWeldStart)
      { S7_Templates := "SrcType := LReal" } LT_Contact(in1 := #Torch.COut.ActualPosition, in2 := #Sts.WeldCycle.PosWeldStop)
      wire#w5
      Coil( #Sts.Torch.InWeldON )
   END_RUNG
   RUNG wire#powerrail
      I_Contact( #CurrentWeldingSetUp.WeldingDirection )
      { S7_Templates := "SrcType := LReal" } LT_Contact(in1 := #Torch.COut.ActualPosition, in2 := #Sts.WeldCycle.PosWeldStart)
      { S7_Templates := "SrcType := LReal" } GT_Contact(in1 := #Torch.COut.ActualPosition, in2 := #Sts.WeldCycle.PosWeldStop)
   END_RUNG wire#w5
   RUNG wire#powerrail
      { S7_Templates := "SrcType := LReal" } GE_Contact(in1 := #Torch.COut.ActualPosition, in2 := #Sts.WeldCycle.PosMinusInhibit)
      { S7_Templates := "SrcType := LReal" } LE_Contact(in1 := #Torch.COut.ActualPosition, in2 := #Sts.WeldCycle.PosPlusInhibit)
      { S7_Templates := "SrcType := LReal" } GT_Contact(in1 := #PersistentValues.Torch.InhibitWeld_Window, in2 := 0.0)
      Coil( #Sts.Torch.InWeldInhibit )
   END_RUNG
   RUNG wire#powerrail
      Contact( #CurrentWeldingSetUp.WeldingDirection )
      { S7_Templates := "SrcType := LReal" } GT_Contact(in1 := #Torch.COut.ActualPosition, in2 := #Sts.WeldCycle.PosOutStripEdgeSideWeldStart)
      { S7_Templates := "SrcType := LReal" } LT_Contact(in1 := #Torch.COut.ActualPosition, in2 := #Sts.WeldCycle.PosOutStripEdgeSideWeldStop)
      wire#w6
      Coil( #Sts.Torch.InPotentimeterON )
   END_RUNG
   RUNG wire#powerrail
      I_Contact( #CurrentWeldingSetUp.WeldingDirection )
      { S7_Templates := "SrcType := LReal" } LT_Contact(in1 := #Torch.COut.ActualPosition, in2 := #Sts.WeldCycle.PosOutStripEdgeSideWeldStart)
      { S7_Templates := "SrcType := LReal" } GT_Contact(in1 := #Torch.COut.ActualPosition, in2 := #Sts.WeldCycle.PosOutStripEdgeSideWeldStop)
   END_RUNG wire#w6
   RUNG wire#powerrail
      I_Contact( #Sts.WeldCycle.ON1 )
      I_Contact( #Sts.WeldCycle.ON2 )
      Not()
      Contact( #Sts.Torch.InWeldON )
   END_RUNG wire#w6
   // the same network as SCL:
   #PosOK := "TolWindow"(ActPos := #Torch.COut.ActualPosition,
                         Target := #PersistentValues.Torch.Parking_Pos,
                         PosWin := #PersistentValues.TorchAx.PosTolerance);
   #Sts.Torch.InParkPosition := (#Torch.COut.InPosition AND (#Torch.COut.ActualTargetPos = #PersistentValues.Torch.Parking_Pos)) OR (NOT #Torch.COut.InPosition AND #PosOK);
   #PosOK := "TolWindow"(ActPos := #Torch.COut.ActualPosition,
                         Target := #Sts.WeldCycle.PosOutStripEdgeSideWeldStart,
                         PosWin := #PersistentValues.TorchAx.PosTolerance);
   #Sts.Torch.InOutEdgeOfWeldStart := (#Torch.COut.InPosition AND (#Torch.COut.ActualTargetPos = #Sts.WeldCycle.PosOutStripEdgeSideWeldStart)) OR (NOT #Torch.COut.InPosition AND #PosOK);
   #PosOK := "TolWin_REAL"(ActPos := #Torch.COut.ActualPosition,
                           Target := #Sts.WeldCycle.PosWeldStart,
                           PosWin := #PersistentValues.TorchAx.PosTolerance);
   #Sts.Torch.InWeldStart := (#Torch.COut.InPosition AND (#Torch.COut.ActualTargetPos = #Sts.WeldCycle.PosWeldStart)) OR (NOT #Torch.COut.InPosition AND #PosOK);
   #Sts.Torch.inWeldStop := (#CurrentWeldingSetUp.WeldingDirection AND (#Torch.COut.ActualPosition >= #Sts.WeldCycle.PosWeldStop)) OR (NOT #CurrentWeldingSetUp.WeldingDirection AND (#Torch.COut.ActualPosition <= #Sts.WeldCycle.PosWeldStop));
   #Sts.Torch.InWeldON := (#CurrentWeldingSetUp.WeldingDirection AND (#Torch.COut.ActualPosition > #Sts.WeldCycle.PosWeldStart) AND (#Torch.COut.ActualPosition < #Sts.WeldCycle.PosWeldStop)) OR (NOT #CurrentWeldingSetUp.WeldingDirection AND (#Torch.COut.ActualPosition < #Sts.WeldCycle.PosWeldStart) AND (#Torch.COut.ActualPosition > #Sts.WeldCycle.PosWeldStop));
   #Sts.Torch.InWeldInhibit := (#Torch.COut.ActualPosition >= #Sts.WeldCycle.PosMinusInhibit) AND (#Torch.COut.ActualPosition <= #Sts.WeldCycle.PosPlusInhibit) AND (#PersistentValues.Torch.InhibitWeld_Window > 0.0);
   #Sts.Torch.InPotentimeterON := (#CurrentWeldingSetUp.WeldingDirection AND (#Torch.COut.ActualPosition > #Sts.WeldCycle.PosOutStripEdgeSideWeldStart) AND (#Torch.COut.ActualPosition < #Sts.WeldCycle.PosOutStripEdgeSideWeldStop)) OR (NOT #CurrentWeldingSetUp.WeldingDirection AND (#Torch.COut.ActualPosition < #Sts.WeldCycle.PosOutStripEdgeSideWeldStart) AND (#Torch.COut.ActualPosition > #Sts.WeldCycle.PosOutStripEdgeSideWeldStop)) OR (NOT (NOT #Sts.WeldCycle.ON1 AND NOT #Sts.WeldCycle.ON2) AND #Sts.Torch.InWeldON);
END_REGION

REGION Network 23: Reset torch position status if axis is not in operation = hommed
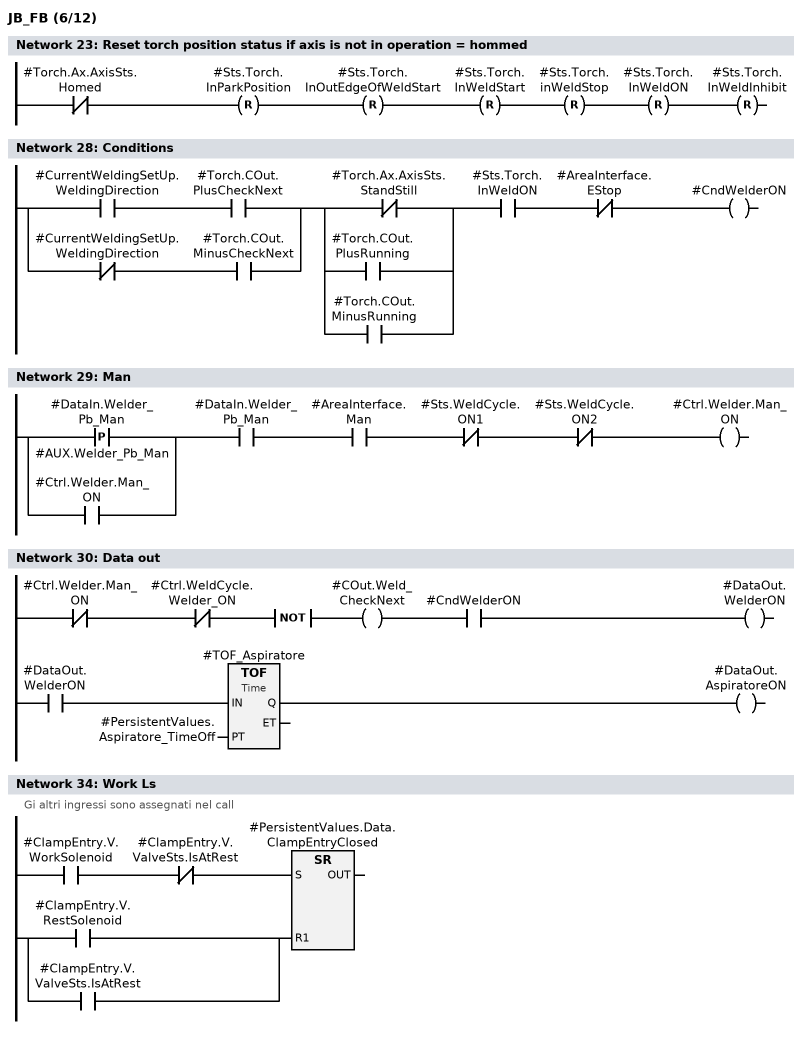
   RUNG wire#powerrail
      I_Contact( #Torch.Ax.AxisSts.Homed )
      R_Coil( #Sts.Torch.InParkPosition )
      R_Coil( #Sts.Torch.InOutEdgeOfWeldStart )
      R_Coil( #Sts.Torch.InWeldStart )
      R_Coil( #Sts.Torch.inWeldStop )
      R_Coil( #Sts.Torch.InWeldON )
      R_Coil( #Sts.Torch.InWeldInhibit )
   END_RUNG
   // the same network as SCL:
   IF NOT #Torch.Ax.AxisSts.Homed THEN
       #Sts.Torch.InParkPosition := FALSE;
       #Sts.Torch.InOutEdgeOfWeldStart := FALSE;
       #Sts.Torch.InWeldStart := FALSE;
       #Sts.Torch.inWeldStop := FALSE;
       #Sts.Torch.InWeldON := FALSE;
       #Sts.Torch.InWeldInhibit := FALSE;
   END_IF;
END_REGION

REGION Network 24: >
END_REGION

REGION Network 25: >
END_REGION

REGION Network 26: >
END_REGION

REGION Network 27: <<< WELDER >>
END_REGION

REGION Network 28: Conditions
   RUNG wire#powerrail
      Contact( #CurrentWeldingSetUp.WeldingDirection )
      Contact( #Torch.COut.PlusCheckNext )
      wire#w1
      I_Contact( #Torch.Ax.AxisSts.StandStill )
      wire#w2
      Contact( #Sts.Torch.InWeldON )
      I_Contact( #AreaInterface.EStop )
      Coil( #CndWelderON )
   END_RUNG
   RUNG wire#powerrail
      I_Contact( #CurrentWeldingSetUp.WeldingDirection )
      Contact( #Torch.COut.MinusCheckNext )
   END_RUNG wire#w1
   RUNG wire#w1
      Contact( #Torch.COut.PlusRunning )
   END_RUNG wire#w2
   RUNG wire#w1
      Contact( #Torch.COut.MinusRunning )
   END_RUNG wire#w2
   // the same network as SCL:
   #CndWelderON := ((#CurrentWeldingSetUp.WeldingDirection AND #Torch.COut.PlusCheckNext) OR (NOT #CurrentWeldingSetUp.WeldingDirection AND #Torch.COut.MinusCheckNext)) AND (NOT #Torch.Ax.AxisSts.StandStill OR #Torch.COut.PlusRunning OR #Torch.COut.MinusRunning) AND #Sts.Torch.InWeldON AND NOT #AreaInterface.EStop;
END_REGION

REGION Network 29: Man
   RUNG wire#powerrail
      P_Contact(operand := #DataIn.Welder_Pb_Man, bit := #AUX.Welder_Pb_Man)
      wire#w1
      Contact( #DataIn.Welder_Pb_Man )
      Contact( #AreaInterface.Man )
      I_Contact( #Sts.WeldCycle.ON1 )
      I_Contact( #Sts.WeldCycle.ON2 )
      Coil( #Ctrl.Welder.Man_ON )
   END_RUNG
   RUNG wire#powerrail
      Contact( #Ctrl.Welder.Man_ON )
   END_RUNG wire#w1
   // the same network as SCL:
   #_w1 := #DataIn.Welder_Pb_Man AND NOT #AUX.Welder_Pb_Man;   // rising edge of #DataIn.Welder_Pb_Man
   #AUX.Welder_Pb_Man := #DataIn.Welder_Pb_Man;
   #Ctrl.Welder.Man_ON := (#_w1 OR #Ctrl.Welder.Man_ON) AND #DataIn.Welder_Pb_Man AND #AreaInterface.Man AND NOT #Sts.WeldCycle.ON1 AND NOT #Sts.WeldCycle.ON2;
END_REGION

REGION Network 30: Data out
   RUNG wire#powerrail
      I_Contact( #Ctrl.Welder.Man_ON )
      I_Contact( #Ctrl.WeldCycle.Welder_ON )
      Not()
      Coil( #COut.Weld_CheckNext )
      Contact( #CndWelderON )
      Coil( #DataOut.WelderON )
   END_RUNG
   RUNG wire#powerrail
      Contact( #DataOut.WelderON )
      { S7_Templates := "time_type := Time" } #TOF_Aspiratore.TOF(pt := #PersistentValues.Aspiratore_TimeOff, et =>)
      Coil( #DataOut.AspiratoreON )
   END_RUNG
   // the same network as SCL:
   #COut.Weld_CheckNext := NOT (NOT #Ctrl.Welder.Man_ON AND NOT #Ctrl.WeldCycle.Welder_ON);
   #DataOut.WelderON := #COut.Weld_CheckNext AND #CndWelderON;
   #TOF_Aspiratore(IN := #DataOut.WelderON, PT := #PersistentValues.Aspiratore_TimeOff);   // TOF
   #DataOut.AspiratoreON := #TOF_Aspiratore.Q;
END_REGION

REGION Network 31: >
END_REGION

REGION Network 32: >
END_REGION

REGION Network 33: <<< CLAMP ENTRY >>>
END_REGION

REGION Network 34: Work Ls
   // Gi altri ingressi sono assegnati nel call
   RUNG wire#powerrail
      Contact( #ClampEntry.V.WorkSolenoid )
      I_Contact( #ClampEntry.V.ValveSts.IsAtRest )
      S_SR(operand := #PersistentValues.Data.ClampEntryClosed, r1 := wire#w1)
   END_RUNG
   RUNG wire#powerrail
      Contact( #ClampEntry.V.RestSolenoid )
   END_RUNG wire#w1
   RUNG wire#powerrail
      Contact( #ClampEntry.V.ValveSts.IsAtRest )
   END_RUNG wire#w1
   // the same network as SCL:
   IF #ClampEntry.V.WorkSolenoid AND NOT #ClampEntry.V.ValveSts.IsAtRest THEN
       #PersistentValues.Data.ClampEntryClosed := TRUE;   // SR flip-flop
   END_IF;
   IF #ClampEntry.V.RestSolenoid OR #ClampEntry.V.ValveSts.IsAtRest THEN
       #PersistentValues.Data.ClampEntryClosed := FALSE;
   END_IF;
END_REGION

REGION Network 35 (SCL): Data in
   #ClampEntry.DataIn := #DataIn.ClampEntry;

   #ClampEntry.DataIn.Work_Ls[1] := #PersistentValues.Data.ClampEntryClosed;
END_REGION

REGION Network 36: CIn (Manager = Welding Cycle)
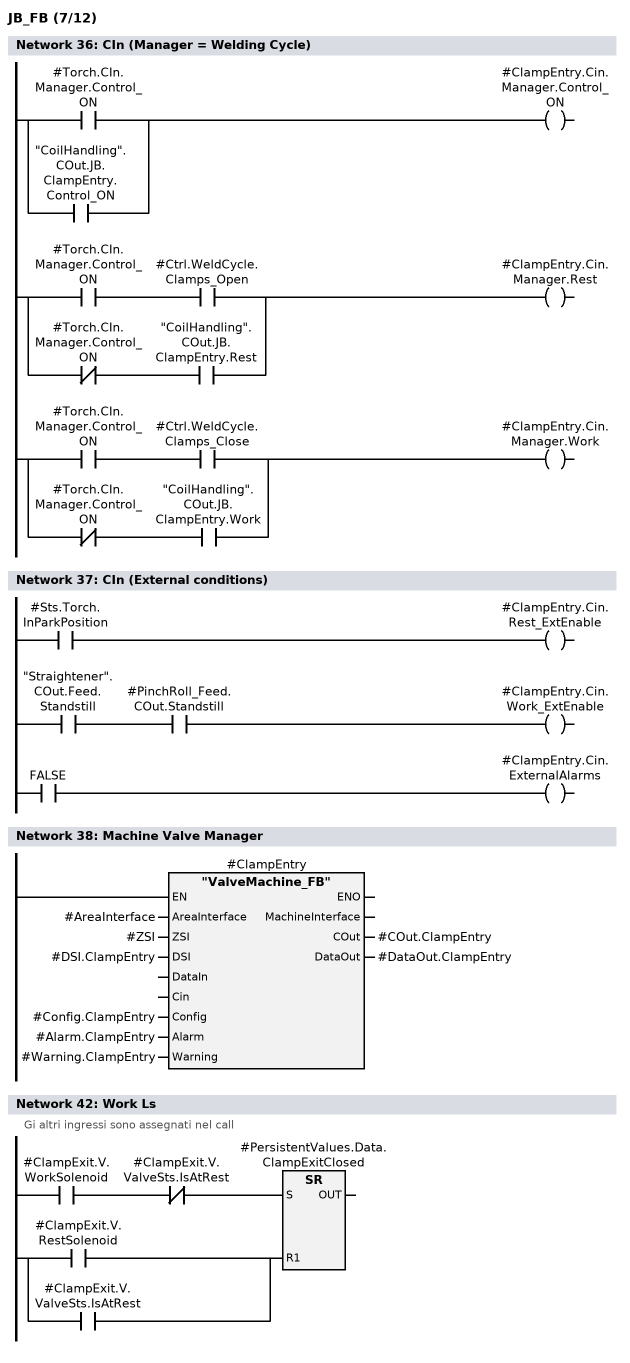
   RUNG wire#powerrail
      Contact( #Torch.CIn.Manager.Control_ON )
      wire#w1
      Coil( #ClampEntry.Cin.Manager.Control_ON )
   END_RUNG
   RUNG wire#powerrail
      Contact( "CoilHandling".COut.JB.ClampEntry.Control_ON )
   END_RUNG wire#w1
   RUNG wire#powerrail
      Contact( #Torch.CIn.Manager.Control_ON )
      Contact( #Ctrl.WeldCycle.Clamps_Open )
      wire#w2
      Coil( #ClampEntry.Cin.Manager.Rest )
   END_RUNG
   RUNG wire#powerrail
      I_Contact( #Torch.CIn.Manager.Control_ON )
      Contact( "CoilHandling".COut.JB.ClampEntry.Rest )
   END_RUNG wire#w2
   RUNG wire#powerrail
      Contact( #Torch.CIn.Manager.Control_ON )
      Contact( #Ctrl.WeldCycle.Clamps_Close )
      wire#w3
      Coil( #ClampEntry.Cin.Manager.Work )
   END_RUNG
   RUNG wire#powerrail
      I_Contact( #Torch.CIn.Manager.Control_ON )
      Contact( "CoilHandling".COut.JB.ClampEntry.Work )
   END_RUNG wire#w3
   // the same network as SCL:
   #ClampEntry.Cin.Manager.Control_ON := #Torch.CIn.Manager.Control_ON OR "CoilHandling".COut.JB.ClampEntry.Control_ON;
   #ClampEntry.Cin.Manager.Rest := (#Torch.CIn.Manager.Control_ON AND #Ctrl.WeldCycle.Clamps_Open) OR (NOT #Torch.CIn.Manager.Control_ON AND "CoilHandling".COut.JB.ClampEntry.Rest);
   #ClampEntry.Cin.Manager.Work := (#Torch.CIn.Manager.Control_ON AND #Ctrl.WeldCycle.Clamps_Close) OR (NOT #Torch.CIn.Manager.Control_ON AND "CoilHandling".COut.JB.ClampEntry.Work);
END_REGION

REGION Network 37: CIn (External conditions)
   RUNG wire#powerrail
      Contact( #Sts.Torch.InParkPosition )
      Coil( #ClampEntry.Cin.Rest_ExtEnable )
   END_RUNG
   RUNG wire#powerrail
      Contact( "Straightener".COut.Feed.Standstill )
      Contact( #PinchRoll_Feed.COut.Standstill )
      Coil( #ClampEntry.Cin.Work_ExtEnable )
   END_RUNG
   RUNG wire#powerrail
      Contact( FALSE )
      Coil( #ClampEntry.Cin.ExternalAlarms )
   END_RUNG
   // the same network as SCL:
   #ClampEntry.Cin.Rest_ExtEnable := #Sts.Torch.InParkPosition;
   #ClampEntry.Cin.Work_ExtEnable := "Straightener".COut.Feed.Standstill AND #PinchRoll_Feed.COut.Standstill;
   #ClampEntry.Cin.ExternalAlarms := FALSE;
END_REGION

REGION Network 38: Machine Valve Manager
   RUNG wire#powerrail
      #ClampEntry(AreaInterface := #AreaInterface, ZSI := #ZSI, DSI := #DSI.ClampEntry, DataIn :=, Cin :=, Config := #Config.ClampEntry, Alarm := #Alarm.ClampEntry, Warning := #Warning.ClampEntry, MachineInterface =>, COut => #COut.ClampEntry, DataOut => #DataOut.ClampEntry)
   END_RUNG
   // the same network as SCL:
   #ClampEntry(AreaInterface := #AreaInterface,   // "ValveMachine_FB"
               ZSI := #ZSI,
               DSI := #DSI.ClampEntry,
               Config := #Config.ClampEntry,
               Alarm := #Alarm.ClampEntry,
               Warning := #Warning.ClampEntry,
               COut => #COut.ClampEntry,
               DataOut => #DataOut.ClampEntry);
END_REGION

REGION Network 39: >
END_REGION

REGION Network 40: >
END_REGION

REGION Network 41: <<< CLAMP EXIT >>>
END_REGION

REGION Network 42: Work Ls
   // Gi altri ingressi sono assegnati nel call
   RUNG wire#powerrail
      Contact( #ClampExit.V.WorkSolenoid )
      I_Contact( #ClampExit.V.ValveSts.IsAtRest )
      S_SR(operand := #PersistentValues.Data.ClampExitClosed, r1 := wire#w1)
   END_RUNG
   RUNG wire#powerrail
      Contact( #ClampExit.V.RestSolenoid )
   END_RUNG wire#w1
   RUNG wire#powerrail
      Contact( #ClampExit.V.ValveSts.IsAtRest )
   END_RUNG wire#w1
   // the same network as SCL:
   IF #ClampExit.V.WorkSolenoid AND NOT #ClampExit.V.ValveSts.IsAtRest THEN
       #PersistentValues.Data.ClampExitClosed := TRUE;   // SR flip-flop
   END_IF;
   IF #ClampExit.V.RestSolenoid OR #ClampExit.V.ValveSts.IsAtRest THEN
       #PersistentValues.Data.ClampExitClosed := FALSE;
   END_IF;
END_REGION

REGION Network 43 (SCL): Data in
   #ClampExit.DataIn := #DataIn.ClampExit;

   #ClampExit.DataIn.Work_Ls[1] := #PersistentValues.Data.ClampExitClosed;
END_REGION

REGION Network 44: CIn (Manager = Welding Cycle)
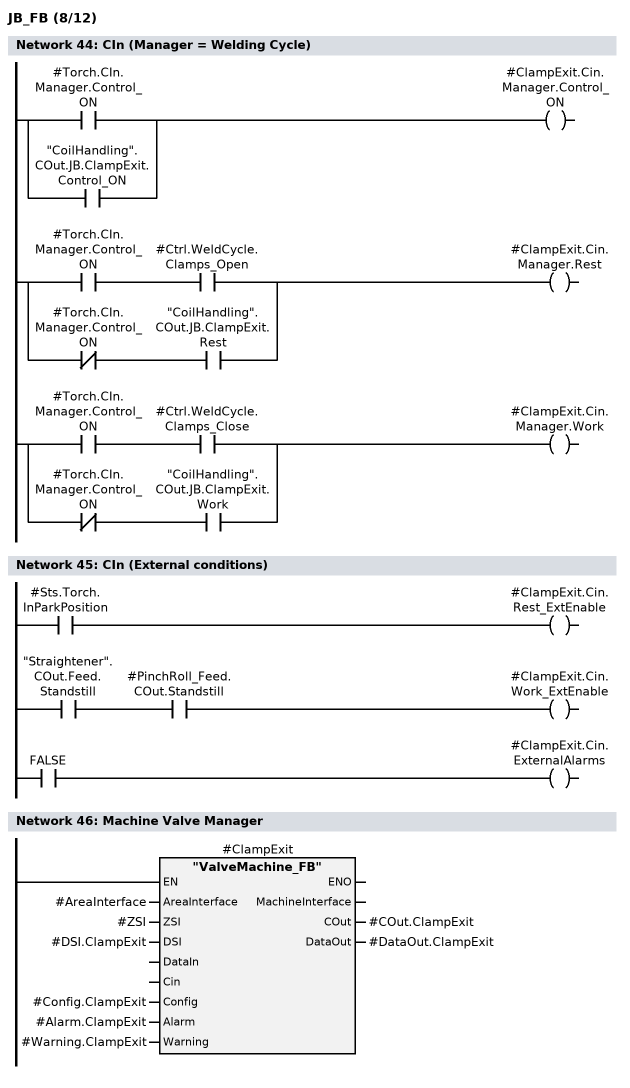
   RUNG wire#powerrail
      Contact( #Torch.CIn.Manager.Control_ON )
      wire#w1
      Coil( #ClampExit.Cin.Manager.Control_ON )
   END_RUNG
   RUNG wire#powerrail
      Contact( "CoilHandling".COut.JB.ClampExit.Control_ON )
   END_RUNG wire#w1
   RUNG wire#powerrail
      Contact( #Torch.CIn.Manager.Control_ON )
      Contact( #Ctrl.WeldCycle.Clamps_Open )
      wire#w2
      Coil( #ClampExit.Cin.Manager.Rest )
   END_RUNG
   RUNG wire#powerrail
      I_Contact( #Torch.CIn.Manager.Control_ON )
      Contact( "CoilHandling".COut.JB.ClampExit.Rest )
   END_RUNG wire#w2
   RUNG wire#powerrail
      Contact( #Torch.CIn.Manager.Control_ON )
      Contact( #Ctrl.WeldCycle.Clamps_Close )
      wire#w3
      Coil( #ClampExit.Cin.Manager.Work )
   END_RUNG
   RUNG wire#powerrail
      I_Contact( #Torch.CIn.Manager.Control_ON )
      Contact( "CoilHandling".COut.JB.ClampExit.Work )
   END_RUNG wire#w3
   // the same network as SCL:
   #ClampExit.Cin.Manager.Control_ON := #Torch.CIn.Manager.Control_ON OR "CoilHandling".COut.JB.ClampExit.Control_ON;
   #ClampExit.Cin.Manager.Rest := (#Torch.CIn.Manager.Control_ON AND #Ctrl.WeldCycle.Clamps_Open) OR (NOT #Torch.CIn.Manager.Control_ON AND "CoilHandling".COut.JB.ClampExit.Rest);
   #ClampExit.Cin.Manager.Work := (#Torch.CIn.Manager.Control_ON AND #Ctrl.WeldCycle.Clamps_Close) OR (NOT #Torch.CIn.Manager.Control_ON AND "CoilHandling".COut.JB.ClampExit.Work);
END_REGION

REGION Network 45: CIn (External conditions)
   RUNG wire#powerrail
      Contact( #Sts.Torch.InParkPosition )
      Coil( #ClampExit.Cin.Rest_ExtEnable )
   END_RUNG
   RUNG wire#powerrail
      Contact( "Straightener".COut.Feed.Standstill )
      Contact( #PinchRoll_Feed.COut.Standstill )
      Coil( #ClampExit.Cin.Work_ExtEnable )
   END_RUNG
   RUNG wire#powerrail
      Contact( FALSE )
      Coil( #ClampExit.Cin.ExternalAlarms )
   END_RUNG
   // the same network as SCL:
   #ClampExit.Cin.Rest_ExtEnable := #Sts.Torch.InParkPosition;
   #ClampExit.Cin.Work_ExtEnable := "Straightener".COut.Feed.Standstill AND #PinchRoll_Feed.COut.Standstill;
   #ClampExit.Cin.ExternalAlarms := FALSE;
END_REGION

REGION Network 46: Machine Valve Manager
   RUNG wire#powerrail
      #ClampExit(AreaInterface := #AreaInterface, ZSI := #ZSI, DSI := #DSI.ClampExit, DataIn :=, Cin :=, Config := #Config.ClampExit, Alarm := #Alarm.ClampExit, Warning := #Warning.ClampExit, MachineInterface =>, COut => #COut.ClampExit, DataOut => #DataOut.ClampExit)
   END_RUNG
   // the same network as SCL:
   #ClampExit(AreaInterface := #AreaInterface,   // "ValveMachine_FB"
              ZSI := #ZSI,
              DSI := #DSI.ClampExit,
              Config := #Config.ClampExit,
              Alarm := #Alarm.ClampExit,
              Warning := #Warning.ClampExit,
              COut => #COut.ClampExit,
              DataOut => #DataOut.ClampExit);
END_REGION

REGION Network 47: >
END_REGION

REGION Network 48: >
END_REGION

REGION Network 49: Sequence of a manual cut cycle
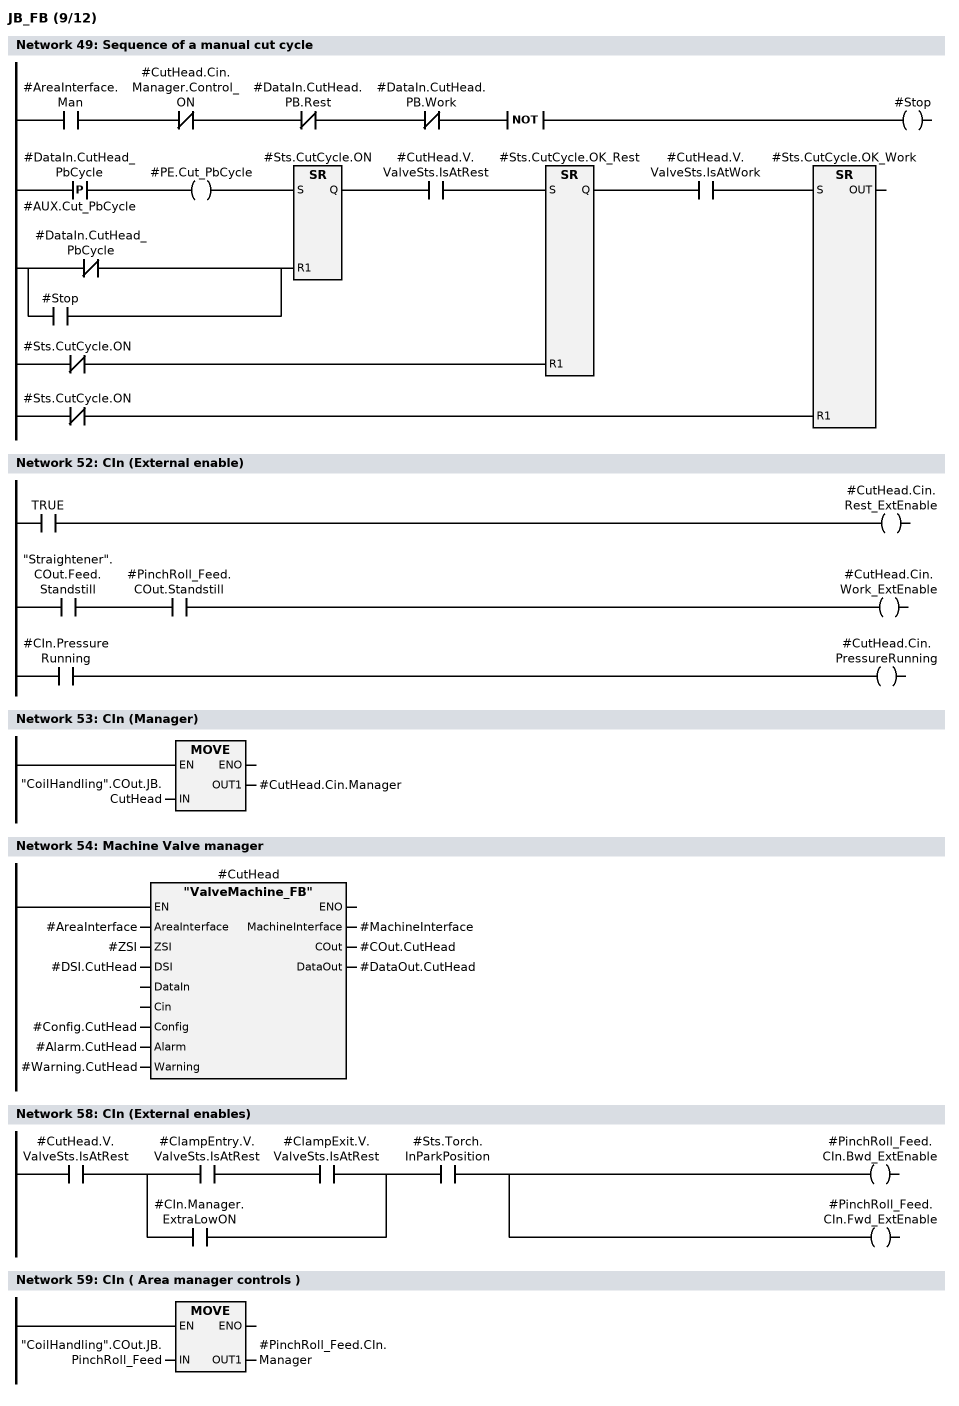
   RUNG wire#powerrail
      Contact( #AreaInterface.Man )
      I_Contact( #CutHead.Cin.Manager.Control_ON )
      I_Contact( #DataIn.CutHead.PB.Rest )
      I_Contact( #DataIn.CutHead.PB.Work )
      Not()
      Coil( #Stop )
   END_RUNG
   RUNG wire#powerrail
      P_Contact(operand := #DataIn.CutHead_PbCycle, bit := #AUX.Cut_PbCycle)
      Coil( #PE.Cut_PbCycle )
      S_SR(operand := #Sts.CutCycle.ON, r1 := wire#w1)
      Contact( #CutHead.V.ValveSts.IsAtRest )
      S_SR(operand := #Sts.CutCycle.OK_Rest, r1 := wire#w2)
      Contact( #CutHead.V.ValveSts.IsAtWork )
      S_SR(operand := #Sts.CutCycle.OK_Work, r1 := wire#w3)
   END_RUNG
   RUNG wire#powerrail
      I_Contact( #DataIn.CutHead_PbCycle )
   END_RUNG wire#w1
   RUNG wire#powerrail
      Contact( #Stop )
   END_RUNG wire#w1
   RUNG wire#powerrail
      I_Contact( #Sts.CutCycle.ON )
   END_RUNG wire#w2
   RUNG wire#powerrail
      I_Contact( #Sts.CutCycle.ON )
   END_RUNG wire#w3
   // the same network as SCL:
   #Stop := NOT (#AreaInterface.Man AND NOT #CutHead.Cin.Manager.Control_ON AND NOT #DataIn.CutHead.PB.Rest AND NOT #DataIn.CutHead.PB.Work);
   #_w1 := #DataIn.CutHead_PbCycle AND NOT #AUX.Cut_PbCycle;   // rising edge of #DataIn.CutHead_PbCycle
   #AUX.Cut_PbCycle := #DataIn.CutHead_PbCycle;
   #PE.Cut_PbCycle := #_w1;
   IF #_w1 THEN
       #Sts.CutCycle.ON := TRUE;   // SR flip-flop
   END_IF;
   IF NOT #DataIn.CutHead_PbCycle OR #Stop THEN #Sts.CutCycle.ON := FALSE; END_IF;
   IF #Sts.CutCycle.ON AND #CutHead.V.ValveSts.IsAtRest THEN
       #Sts.CutCycle.OK_Rest := TRUE;   // SR flip-flop
   END_IF;
   IF NOT #Sts.CutCycle.ON THEN #Sts.CutCycle.OK_Rest := FALSE; END_IF;
   IF #Sts.CutCycle.OK_Rest AND #CutHead.V.ValveSts.IsAtWork THEN
       #Sts.CutCycle.OK_Work := TRUE;   // SR flip-flop
   END_IF;
   IF NOT #Sts.CutCycle.ON THEN #Sts.CutCycle.OK_Work := FALSE; END_IF;
END_REGION

REGION Network 50: <<< CUT HEAD >>
END_REGION

REGION Network 51 (SCL): Data in
   #CutHead.DataIn := #DataIn.CutHead;

   IF #Sts.CutCycle.ON AND
       (NOT #Sts.CutCycle.OK_Rest OR
       (#Sts.CutCycle.OK_Work AND NOT #CutHead.Ctrl.Work_Man))
   THEN
       #CutHead.DataIn.PB.Rest := NOT #CutHead.Ctrl.Work_Man;
   ELSIF #Sts.CutCycle.ON AND
       NOT #Sts.CutCycle.OK_Work
   THEN
       #CutHead.DataIn.PB.Work := TRUE;
   END_IF;
END_REGION

REGION Network 52: CIn (External enable)
   RUNG wire#powerrail
      Contact( TRUE )
      Coil( #CutHead.Cin.Rest_ExtEnable )
   END_RUNG
   RUNG wire#powerrail
      Contact( "Straightener".COut.Feed.Standstill )
      Contact( #PinchRoll_Feed.COut.Standstill )
      Coil( #CutHead.Cin.Work_ExtEnable )
   END_RUNG
   RUNG wire#powerrail
      Contact( #CIn.PressureRunning )
      Coil( #CutHead.Cin.PressureRunning )
   END_RUNG
   // the same network as SCL:
   #CutHead.Cin.Rest_ExtEnable := TRUE;
   #CutHead.Cin.Work_ExtEnable := "Straightener".COut.Feed.Standstill AND #PinchRoll_Feed.COut.Standstill;
   #CutHead.Cin.PressureRunning := #CIn.PressureRunning;
END_REGION

REGION Network 53: CIn (Manager)
   RUNG wire#powerrail
      { S7_GenerateENO := "TRUE" } Move(in := "CoilHandling".COut.JB.CutHead, out1 => #CutHead.Cin.Manager)
   END_RUNG
   // the same network as SCL:
   #CutHead.Cin.Manager := "CoilHandling".COut.JB.CutHead;
END_REGION

REGION Network 54: Machine Valve manager
   RUNG wire#powerrail
      #CutHead(AreaInterface := #AreaInterface, ZSI := #ZSI, DSI := #DSI.CutHead, DataIn :=, Cin :=, Config := #Config.CutHead, Alarm := #Alarm.CutHead, Warning := #Warning.CutHead, MachineInterface => #MachineInterface, COut => #COut.CutHead, DataOut => #DataOut.CutHead)
   END_RUNG
   // the same network as SCL:
   #CutHead(AreaInterface := #AreaInterface,   // "ValveMachine_FB"
            ZSI := #ZSI,
            DSI := #DSI.CutHead,
            Config := #Config.CutHead,
            Alarm := #Alarm.CutHead,
            Warning := #Warning.CutHead,
            MachineInterface => #MachineInterface,
            COut => #COut.CutHead,
            DataOut => #DataOut.CutHead);
END_REGION

REGION Network 55: >
END_REGION

REGION Network 56: >
END_REGION

REGION Network 57: <<< FEED >>>
END_REGION

REGION Network 58: CIn (External enables)
   RUNG wire#powerrail
      Contact( #CutHead.V.ValveSts.IsAtRest )
      wire#w1
      Contact( #ClampEntry.V.ValveSts.IsAtRest )
      Contact( #ClampExit.V.ValveSts.IsAtRest )
      wire#w2
      Contact( #Sts.Torch.InParkPosition )
      wire#w3
      Coil( #PinchRoll_Feed.CIn.Bwd_ExtEnable )
   END_RUNG
   RUNG wire#w1
      Contact( #CIn.Manager.ExtraLowON )
   END_RUNG wire#w2
   RUNG wire#w3
      Coil( #PinchRoll_Feed.CIn.Fwd_ExtEnable )
   END_RUNG
   // the same network as SCL:
   #PinchRoll_Feed.CIn.Bwd_ExtEnable := #CutHead.V.ValveSts.IsAtRest AND ((#ClampEntry.V.ValveSts.IsAtRest AND #ClampExit.V.ValveSts.IsAtRest) OR #CIn.Manager.ExtraLowON) AND #Sts.Torch.InParkPosition;
   #PinchRoll_Feed.CIn.Fwd_ExtEnable := #PinchRoll_Feed.CIn.Bwd_ExtEnable;
END_REGION

REGION Network 59: CIn ( Area manager controls )
   RUNG wire#powerrail
      { S7_GenerateENO := "TRUE" } Move(in := "CoilHandling".COut.JB.PinchRoll_Feed, out1 => #PinchRoll_Feed.CIn.Manager)
   END_RUNG
   // the same network as SCL:
   #PinchRoll_Feed.CIn.Manager := "CoilHandling".COut.JB.PinchRoll_Feed;
END_REGION

REGION Network 60: CIn (Velocity override) when extra low selected
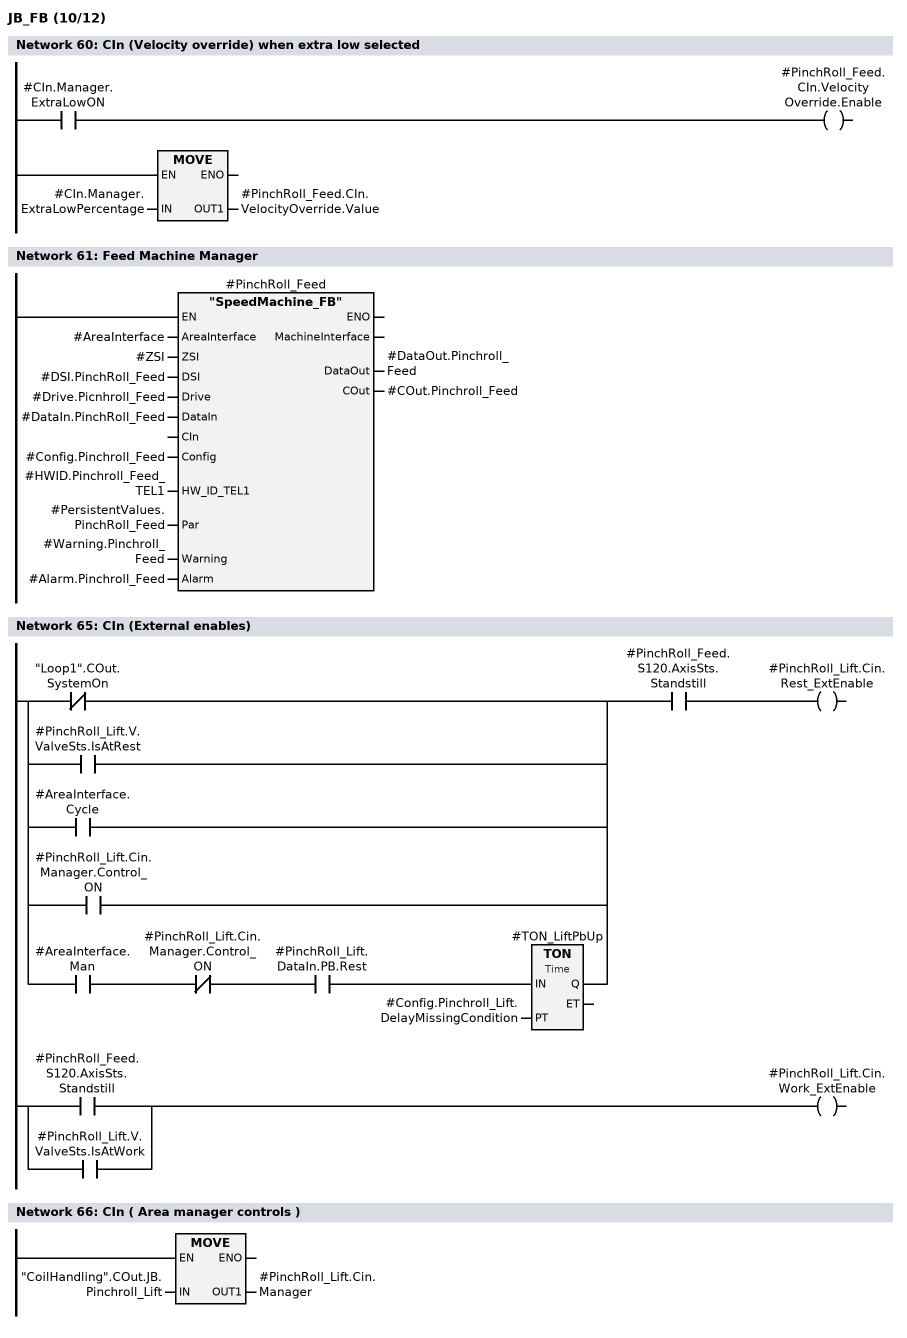
   RUNG wire#powerrail
      Contact( #CIn.Manager.ExtraLowON )
      Coil( #PinchRoll_Feed.CIn.VelocityOverride.Enable )
   END_RUNG
   RUNG wire#powerrail
      { S7_GenerateENO := "TRUE" } Move(in := #CIn.Manager.ExtraLowPercentage, out1 => #PinchRoll_Feed.CIn.VelocityOverride.Value)
   END_RUNG
   // the same network as SCL:
   #PinchRoll_Feed.CIn.VelocityOverride.Enable := #CIn.Manager.ExtraLowON;
   #PinchRoll_Feed.CIn.VelocityOverride.Value := #CIn.Manager.ExtraLowPercentage;
END_REGION

REGION Network 61: Feed Machine Manager
   RUNG wire#powerrail
      #PinchRoll_Feed(AreaInterface := #AreaInterface, ZSI := #ZSI, DSI := #DSI.PinchRoll_Feed, Drive := #Drive.Picnhroll_Feed, DataIn := #DataIn.PinchRoll_Feed, CIn :=, Config := #Config.Pinchroll_Feed, HW_ID_TEL1 := #HWID.Pinchroll_Feed_TEL1, Par := #PersistentValues.PinchRoll_Feed, Warning := #Warning.Pinchroll_Feed, Alarm := #Alarm.Pinchroll_Feed, MachineInterface =>, DataOut => #DataOut.Pinchroll_Feed, COut => #COut.Pinchroll_Feed)
   END_RUNG
   // the same network as SCL:
   #PinchRoll_Feed(AreaInterface := #AreaInterface,   // "SpeedMachine_FB"
                   ZSI := #ZSI,
                   DSI := #DSI.PinchRoll_Feed,
                   Drive := #Drive.Picnhroll_Feed,
                   DataIn := #DataIn.PinchRoll_Feed,
                   Config := #Config.Pinchroll_Feed,
                   HW_ID_TEL1 := #HWID.Pinchroll_Feed_TEL1,
                   Par := #PersistentValues.PinchRoll_Feed,
                   Warning := #Warning.Pinchroll_Feed,
                   Alarm := #Alarm.Pinchroll_Feed,
                   DataOut => #DataOut.Pinchroll_Feed,
                   COut => #COut.Pinchroll_Feed);
END_REGION

REGION Network 62: >
END_REGION

REGION Network 63: >
END_REGION

REGION Network 64: <<< LIFT >>>
END_REGION

REGION Network 65: CIn (External enables)
   RUNG wire#powerrail
      I_Contact( "Loop1".COut.SystemOn )
      wire#w1
      Contact( #PinchRoll_Feed.S120.AxisSts.Standstill )
      Coil( #PinchRoll_Lift.Cin.Rest_ExtEnable )
   END_RUNG
   RUNG wire#powerrail
      Contact( #PinchRoll_Lift.V.ValveSts.IsAtRest )
   END_RUNG wire#w1
   RUNG wire#powerrail
      Contact( #AreaInterface.Cycle )
   END_RUNG wire#w1
   RUNG wire#powerrail
      Contact( #PinchRoll_Lift.Cin.Manager.Control_ON )
   END_RUNG wire#w1
   RUNG wire#powerrail
      Contact( #AreaInterface.Man )
      I_Contact( #PinchRoll_Lift.Cin.Manager.Control_ON )
      Contact( #PinchRoll_Lift.DataIn.PB.Rest )
      { S7_Templates := "time_type := Time" } #TON_LiftPbUp.TON(pt := #Config.Pinchroll_Lift.DelayMissingCondition, et =>)
   END_RUNG wire#w1
   RUNG wire#powerrail
      Contact( #PinchRoll_Feed.S120.AxisSts.Standstill )
      wire#w2
      Coil( #PinchRoll_Lift.Cin.Work_ExtEnable )
   END_RUNG
   RUNG wire#powerrail
      Contact( #PinchRoll_Lift.V.ValveSts.IsAtWork )
   END_RUNG wire#w2
   // the same network as SCL:
   #TON_LiftPbUp(IN := #AreaInterface.Man AND NOT #PinchRoll_Lift.Cin.Manager.Control_ON AND #PinchRoll_Lift.DataIn.PB.Rest,   // TON
                 PT := #Config.Pinchroll_Lift.DelayMissingCondition);
   #PinchRoll_Lift.Cin.Rest_ExtEnable := (NOT "Loop1".COut.SystemOn OR #PinchRoll_Lift.V.ValveSts.IsAtRest OR #AreaInterface.Cycle OR #PinchRoll_Lift.Cin.Manager.Control_ON OR #TON_LiftPbUp.Q) AND #PinchRoll_Feed.S120.AxisSts.Standstill;
   #PinchRoll_Lift.Cin.Work_ExtEnable := #PinchRoll_Feed.S120.AxisSts.Standstill OR #PinchRoll_Lift.V.ValveSts.IsAtWork;
END_REGION

REGION Network 66: CIn ( Area manager controls )
   RUNG wire#powerrail
      { S7_GenerateENO := "TRUE" } Move(in := "CoilHandling".COut.JB.Pinchroll_Lift, out1 => #PinchRoll_Lift.Cin.Manager)
   END_RUNG
   // the same network as SCL:
   #PinchRoll_Lift.Cin.Manager := "CoilHandling".COut.JB.Pinchroll_Lift;
END_REGION

REGION Network 67: Valve machine Manager
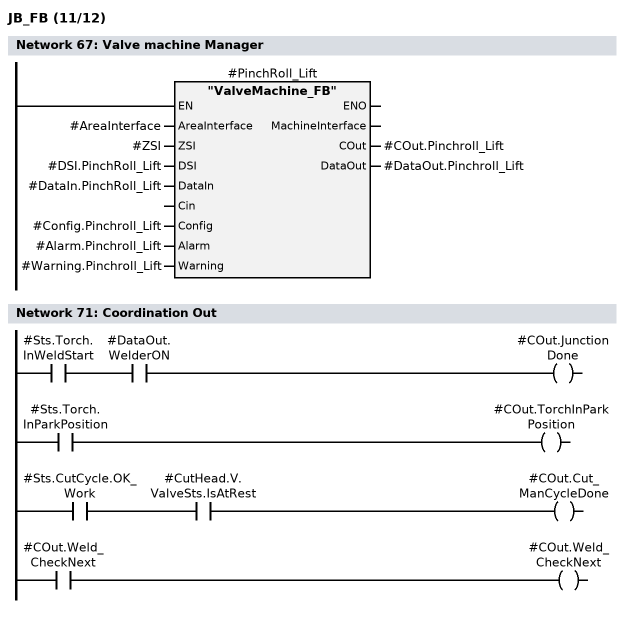
   RUNG wire#powerrail
      #PinchRoll_Lift(AreaInterface := #AreaInterface, ZSI := #ZSI, DSI := #DSI.PinchRoll_Lift, DataIn := #DataIn.PinchRoll_Lift, Cin :=, Config := #Config.Pinchroll_Lift, Alarm := #Alarm.Pinchroll_Lift, Warning := #Warning.Pinchroll_Lift, MachineInterface =>, COut => #COut.Pinchroll_Lift, DataOut => #DataOut.Pinchroll_Lift)
   END_RUNG
   // the same network as SCL:
   #PinchRoll_Lift(AreaInterface := #AreaInterface,   // "ValveMachine_FB"
                   ZSI := #ZSI,
                   DSI := #DSI.PinchRoll_Lift,
                   DataIn := #DataIn.PinchRoll_Lift,
                   Config := #Config.Pinchroll_Lift,
                   Alarm := #Alarm.Pinchroll_Lift,
                   Warning := #Warning.Pinchroll_Lift,
                   COut => #COut.Pinchroll_Lift,
                   DataOut => #DataOut.Pinchroll_Lift);
END_REGION

REGION Network 68: >
END_REGION

REGION Network 69: >
END_REGION

REGION Network 70: <<< MACHINE STATUS >>>
END_REGION

REGION Network 71: Coordination Out
   RUNG wire#powerrail
      Contact( #Sts.Torch.InWeldStart )
      Contact( #DataOut.WelderON )
      Coil( #COut.JunctionDone )
   END_RUNG
   RUNG wire#powerrail
      Contact( #Sts.Torch.InParkPosition )
      Coil( #COut.TorchInParkPosition )
   END_RUNG
   RUNG wire#powerrail
      Contact( #Sts.CutCycle.OK_Work )
      Contact( #CutHead.V.ValveSts.IsAtRest )
      Coil( #COut.Cut_ManCycleDone )
   END_RUNG
   RUNG wire#powerrail
      Contact( #COut.Weld_CheckNext )
      Coil( #COut.Weld_CheckNext )
   END_RUNG
   // the same network as SCL:
   #COut.JunctionDone := #Sts.Torch.InWeldStart AND #DataOut.WelderON;
   #COut.TorchInParkPosition := #Sts.Torch.InParkPosition;
   #COut.Cut_ManCycleDone := #Sts.CutCycle.OK_Work AND #CutHead.V.ValveSts.IsAtRest;
   #COut.Weld_CheckNext := #COut.Weld_CheckNext;
END_REGION

REGION Network 72: Collect machine to zone interface (internal machines OR)
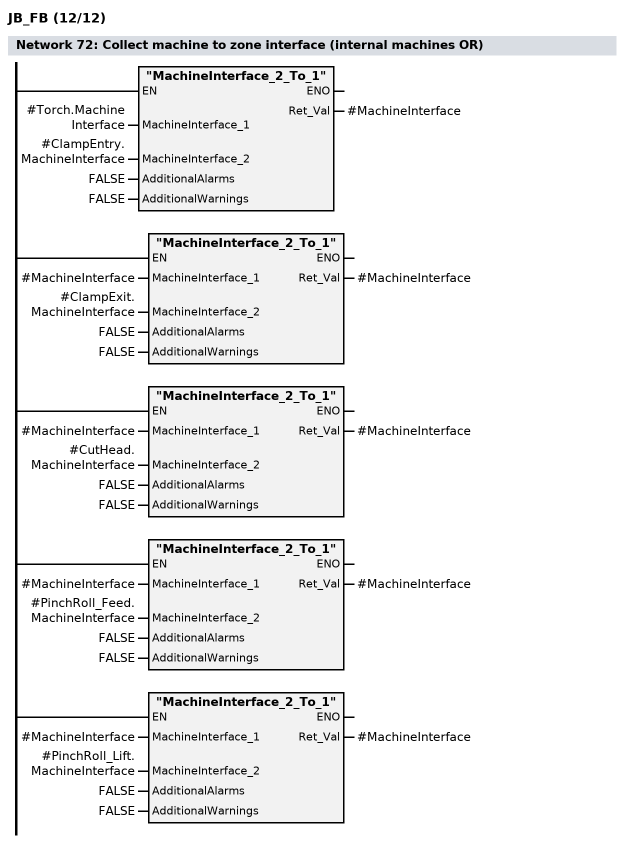
   RUNG wire#powerrail
      "MachineInterface_2_To_1"(MachineInterface_1 := #Torch.MachineInterface, MachineInterface_2 := #ClampEntry.MachineInterface, AdditionalAlarms := FALSE, AdditionalWarnings := FALSE, Ret_Val => #MachineInterface)
   END_RUNG
   RUNG wire#powerrail
      "MachineInterface_2_To_1"(MachineInterface_1 := #MachineInterface, MachineInterface_2 := #ClampExit.MachineInterface, AdditionalAlarms := FALSE, AdditionalWarnings := FALSE, Ret_Val => #MachineInterface)
   END_RUNG
   RUNG wire#powerrail
      "MachineInterface_2_To_1"(MachineInterface_1 := #MachineInterface, MachineInterface_2 := #CutHead.MachineInterface, AdditionalAlarms := FALSE, AdditionalWarnings := FALSE, Ret_Val => #MachineInterface)
   END_RUNG
   RUNG wire#powerrail
      "MachineInterface_2_To_1"(MachineInterface_1 := #MachineInterface, MachineInterface_2 := #PinchRoll_Feed.MachineInterface, AdditionalAlarms := FALSE, AdditionalWarnings := FALSE, Ret_Val => #MachineInterface)
   END_RUNG
   RUNG wire#powerrail
      "MachineInterface_2_To_1"(MachineInterface_1 := #MachineInterface, MachineInterface_2 := #PinchRoll_Lift.MachineInterface, AdditionalAlarms := FALSE, AdditionalWarnings := FALSE, Ret_Val => #MachineInterface)
   END_RUNG
   // the same network as SCL:
   #MachineInterface := "MachineInterface_2_To_1"(MachineInterface_1 := #Torch.MachineInterface,
                           MachineInterface_2 := #ClampEntry.MachineInterface,
                           AdditionalAlarms := FALSE,
                           AdditionalWarnings := FALSE);
   #MachineInterface := "MachineInterface_2_To_1"(MachineInterface_1 := #MachineInterface,
                           MachineInterface_2 := #ClampExit.MachineInterface,
                           AdditionalAlarms := FALSE,
                           AdditionalWarnings := FALSE);
   #MachineInterface := "MachineInterface_2_To_1"(MachineInterface_1 := #MachineInterface,
                           MachineInterface_2 := #CutHead.MachineInterface,
                           AdditionalAlarms := FALSE,
                           AdditionalWarnings := FALSE);
   #MachineInterface := "MachineInterface_2_To_1"(MachineInterface_1 := #MachineInterface,
                           MachineInterface_2 := #PinchRoll_Feed.MachineInterface,
                           AdditionalAlarms := FALSE,
                           AdditionalWarnings := FALSE);
   #MachineInterface := "MachineInterface_2_To_1"(MachineInterface_1 := #MachineInterface,
                           MachineInterface_2 := #PinchRoll_Lift.MachineInterface,
                           AdditionalAlarms := FALSE,
                           AdditionalWarnings := FALSE);
END_REGION

REGION Network 73: >
END_REGION

REGION Network 74: >
END_REGION
END_FUNCTION_BLOCK
